LIN {X 0.039,Y -397.005,Z 723.798,A 0.000,B 0.000,C 90.000,E1 179.599} C_DIS
LIN {X 0.011,Y -394.562,Z 723.784,A 0.000,B 0.000,C 90.000,E1 177.135} C_DIS
LIN {X -0.144,Y -391.958,Z 723.766,A 0.000,B 0.000,C 90.000,E1 173.970} C_DIS
LIN {X 0.090,Y -389.994,Z 723.749,A 0.000,B 0.000,C 90.000,E1 170.735} C_DIS
LIN {X -0.181,Y -389.319,Z 723.739,A 0.000,B 0.000,C 90.000,E1 168.993} C_DIS
LIN {X 0.066,Y -388.633,Z 723.729,A 0.000,B 0.000,C 90.000,E1 167.173} C_DIS
LIN {X -0.020,Y -387.919,Z 723.715,A 0.000,B 0.000,C 90.000,E1 164.685} C_DIS
LIN {X -0.021,Y -387.556,Z 723.701,A 0.000,B 0.000,C 90.000,E1 162.181} C_DIS
LIN {X -0.174,Y -387.268,Z 723.687,A 0.000,B 0.000,C 90.000,E1 159.699} C_DIS
LIN {X -0.072,Y -387.127,Z 723.673,A 0.000,B 0.000,C 90.000,E1 157.177} C_DIS
LIN {X -0.029,Y -387.222,Z 723.659,A 0.000,B 0.000,C 90.000,E1 154.665} C_DIS
LIN {X 0.188,Y -387.591,Z 723.643,A 0.000,B 0.000,C 90.000,E1 151.769} C_DIS
LIN {X -0.098,Y -388.115,Z 723.631,A 0.000,B 0.000,C 90.000,E1 149.665} C_DIS
LIN {X 0.077,Y -392.344,Z 723.598,A 0.000,B 0.000,C 90.000,E1 143.577} C_DIS
LIN {X 0.120,Y -395.287,Z 723.584,A 0.000,B 0.000,C 90.000,E1 141.090} C_DIS
LIN {X 0.042,Y -398.011,Z 723.574,A 0.000,B 0.000,C 90.000,E1 139.337} C_DIS
LIN {X -0.158,Y -398.633,Z 723.572,A 0.000,B 0.000,C 90.000,E1 139.013} C_DIS
LIN {X 0.127,Y -401.198,Z 723.566,A 0.000,B 0.000,C 90.000,E1 137.919} C_DIS
LIN {X 0.148,Y -402.865,Z 723.563,A 0.000,B 0.000,C 90.000,E1 137.391} C_DIS
LIN {X -0.092,Y -405.391,Z 723.560,A 0.000,B 0.000,C 90.000,E1 136.863} C_DIS
LIN {X 0.231,Y -408.949,Z 723.557,A 0.000,B 0.000,C 90.000,E1 136.296} C_DIS
LIN {X 0.266,Y -413.856,Z 723.554,A 0.000,B 0.000,C 90.000,E1 135.729} C_DIS
LIN {X 0.176,Y -435.943,Z 723.542,A 0.000,B 0.000,C 90.000,E1 133.542} C_DIS
LIN {X 0.080,Y -449.355,Z 723.535,A 0.000,B 0.000,C 90.000,E1 132.324} C_DIS
LIN {X 0.027,Y -458.279,Z 723.531,A 0.000,B 0.000,C 90.000,E1 131.515} C_DIS
LIN {X -0.130,Y -467.101,Z 723.526,A 0.000,B 0.000,C 90.000,E1 130.701} C_DIS
LIN {X -0.097,Y -474.239,Z 723.522,A 0.000,B 0.000,C 90.000,E1 130.011} C_DIS
LIN {X 0.038,Y -482.703,Z 723.518,A 0.000,B 0.000,C 90.000,E1 129.152} C_DIS
LIN {X -0.057,Y -489.338,Z 723.514,A 0.000,B 0.000,C 90.000,E1 128.463} C_DIS
LIN {X -0.026,Y -496.017,Z 723.510,A 0.000,B 0.000,C 90.000,E1 127.729} C_DIS
LIN {X 0.160,Y -505.000,Z 723.504,A 0.000,B 0.000,C 90.000,E1 126.664} C_DIS
LIN {X 0.076,Y -510.728,Z 723.500,A 0.000,B 0.000,C 90.000,E1 125.931} C_DIS
LIN {X -0.208,Y -513.989,Z 723.497,A 0.000,B 0.000,C 90.000,E1 125.518} C_DIS
LIN {X 0.062,Y -522.250,Z 723.490,A 0.000,B 0.000,C 90.000,E1 124.199} C_DIS
LIN {X -0.204,Y -526.316,Z 723.486,A 0.000,B 0.000,C 90.000,E1 123.499} C_DIS
LIN {X 0.008,Y -530.042,Z 723.482,A 0.000,B 0.000,C 90.000,E1 122.752} C_DIS
LIN {X 0.256,Y -533.521,Z 723.478,A 0.000,B 0.000,C 90.000,E1 122.005} C_DIS
LIN {X -0.198,Y -536.730,Z 723.474,A 0.000,B 0.000,C 90.000,E1 121.337} C_DIS
LIN {X -0.303,Y -541.523,Z 723.468,A 0.000,B 0.000,C 90.000,E1 120.207} C_DIS
LIN {X -0.217,Y -545.563,Z 723.462,A 0.000,B 0.000,C 90.000,E1 119.205} C_DIS
LIN {X 0.272,Y -549.894,Z 723.456,A 0.000,B 0.000,C 90.000,E1 118.025} C_DIS
LIN {X 0.056,Y -552.912,Z 723.451,A 0.000,B 0.000,C 90.000,E1 117.206} C_DIS
LIN {X 0.126,Y -555.717,Z 723.447,A 0.000,B 0.000,C 90.000,E1 116.360} C_DIS
LIN {X -0.023,Y -558.233,Z 723.442,A 0.000,B 0.000,C 90.000,E1 115.540} C_DIS
LIN {X -0.142,Y -560.406,Z 723.437,A 0.000,B 0.000,C 90.000,E1 114.719} C_DIS
LIN {X -0.239,Y -562.322,Z 723.433,A 0.000,B 0.000,C 90.000,E1 113.898} C_DIS
LIN {X 0.200,Y -564.005,Z 723.428,A 0.000,B 0.000,C 90.000,E1 113.025} C_DIS
LIN {X 0.134,Y -565.434,Z 723.423,A 0.000,B 0.000,C 90.000,E1 112.206} C_DIS
LIN {X 0.007,Y -567.636,Z 723.416,A 0.000,B 0.000,C 90.000,E1 110.844} C_DIS
LIN {X 0.250,Y -569.725,Z 723.408,A 0.000,B 0.000,C 90.000,E1 109.450} C_DIS
LIN {X -0.187,Y -571.772,Z 723.401,A 0.000,B 0.000,C 90.000,E1 108.127} C_DIS
LIN {X 0.128,Y -573.658,Z 723.393,A 0.000,B 0.000,C 90.000,E1 106.732} C_DIS
LIN {X -0.210,Y -575.815,Z 723.384,A 0.000,B 0.000,C 90.000,E1 105.134} C_DIS
LIN {X 0.202,Y -577.226,Z 723.378,A 0.000,B 0.000,C 90.000,E1 104.008} C_DIS
LIN {X 0.156,Y -579.651,Z 723.367,A 0.000,B 0.000,C 90.000,E1 102.119} C_DIS
LIN {X 0.032,Y -581.442,Z 723.360,A 0.000,B 0.000,C 90.000,E1 100.782} C_DIS
LIN {X -0.051,Y -583.109,Z 723.352,A 0.000,B 0.000,C 90.000,E1 99.443} C_DIS
LIN {X 0.230,Y -584.312,Z 723.346,A 0.000,B 0.000,C 90.000,E1 98.341} C_DIS
LIN {X -0.234,Y -585.981,Z 723.338,A 0.000,B 0.000,C 90.000,E1 96.777} C_DIS
LIN {X 0.006,Y -587.104,Z 723.332,A 0.000,B 0.000,C 90.000,E1 95.682} C_DIS
LIN {X -0.137,Y -588.453,Z 723.324,A 0.000,B 0.000,C 90.000,E1 94.359} C_DIS
LIN {X -0.264,Y -589.659,Z 723.317,A 0.000,B 0.000,C 90.000,E1 93.037} C_DIS
LIN {X 0.180,Y -590.697,Z 723.309,A 0.000,B 0.000,C 90.000,E1 91.661} C_DIS
LIN {X 0.041,Y -591.560,Z 723.302,A 0.000,B 0.000,C 90.000,E1 90.344} C_DIS
LIN {X -0.082,Y -592.267,Z 723.295,A 0.000,B 0.000,C 90.000,E1 89.026} C_DIS
LIN {X 0.247,Y -592.954,Z 723.284,A 0.000,B 0.000,C 90.000,E1 87.135} C_DIS
LIN {X 0.195,Y -593.220,Z 723.277,A 0.000,B 0.000,C 90.000,E1 85.812} C_DIS
LIN {X 0.157,Y -593.390,Z 723.270,A 0.000,B 0.000,C 90.000,E1 84.489} C_DIS
LIN {X -0.204,Y -593.437,Z 723.261,A 0.000,B 0.000,C 90.000,E1 82.932} C_DIS
LIN {X -0.134,Y -593.361,Z 723.256,A 0.000,B 0.000,C 90.000,E1 82.129} C_DIS
LIN {X -0.028,Y -593.126,Z 723.249,A 0.000,B 0.000,C 90.000,E1 80.792} C_DIS
LIN {X 0.080,Y -592.679,Z 723.242,A 0.000,B 0.000,C 90.000,E1 79.454} C_DIS
LIN {X 0.171,Y -591.925,Z 723.234,A 0.000,B 0.000,C 90.000,E1 78.117} C_DIS
LIN {X -0.117,Y -590.766,Z 723.224,A 0.000,B 0.000,C 90.000,E1 76.284} C_DIS
LIN {X 0.050,Y -589.783,Z 723.216,A 0.000,B 0.000,C 90.000,E1 74.936} C_DIS
LIN {X 0.185,Y -588.443,Z 723.208,A 0.000,B 0.000,C 90.000,E1 73.323} C_DIS
LIN {X -0.361,Y -587.491,Z 723.202,A 0.000,B 0.000,C 90.000,E1 72.308} C_DIS
LIN {X 0.232,Y -586.098,Z 723.194,A 0.000,B 0.000,C 90.000,E1 70.913} C_DIS
LIN {X -0.162,Y -584.968,Z 723.188,A 0.000,B 0.000,C 90.000,E1 69.880} C_DIS
LIN {X -0.167,Y -583.271,Z 723.181,A 0.000,B 0.000,C 90.000,E1 68.539} C_DIS
LIN {X 0.145,Y -581.811,Z 723.175,A 0.000,B 0.000,C 90.000,E1 67.433} C_DIS
LIN {X 0.126,Y -580.195,Z 723.169,A 0.000,B 0.000,C 90.000,E1 66.357} C_DIS
LIN {X 0.096,Y -578.301,Z 723.163,A 0.000,B 0.000,C 90.000,E1 65.281} C_DIS
LIN {X 0.188,Y -576.737,Z 723.158,A 0.000,B 0.000,C 90.000,E1 64.460} C_DIS
LIN {X 0.108,Y -574.431,Z 723.152,A 0.000,B 0.000,C 90.000,E1 63.384} C_DIS
LIN {X 0.149,Y -572.490,Z 723.148,A 0.000,B 0.000,C 90.000,E1 62.564} C_DIS
LIN {X -0.075,Y -570.377,Z 723.143,A 0.000,B 0.000,C 90.000,E1 61.769} C_DIS
LIN {X 0.008,Y -567.228,Z 723.137,A 0.000,B 0.000,C 90.000,E1 60.667} C_DIS
LIN {X -0.261,Y -564.647,Z 723.133,A 0.000,B 0.000,C 90.000,E1 59.871} C_DIS
LIN {X 0.016,Y -560.862,Z 723.126,A 0.000,B 0.000,C 90.000,E1 58.742} C_DIS
LIN {X -0.106,Y -558.780,Z 723.123,A 0.000,B 0.000,C 90.000,E1 58.201} C_DIS
LIN {X -0.242,Y -556.592,Z 723.120,A 0.000,B 0.000,C 90.000,E1 57.661} C_DIS
LIN {X 0.141,Y -552.966,Z 723.116,A 0.000,B 0.000,C 90.000,E1 56.786} C_DIS
LIN {X 0.141,Y -549.488,Z 723.112,A 0.000,B 0.000,C 90.000,E1 56.087} C_DIS
LIN {X 0.218,Y -545.757,Z 723.108,A 0.000,B 0.000,C 90.000,E1 55.388} C_DIS
LIN {X 0.154,Y -541.618,Z 723.104,A 0.000,B 0.000,C 90.000,E1 54.689} C_DIS
LIN {X 0.202,Y -538.072,Z 723.101,A 0.000,B 0.000,C 90.000,E1 54.116} C_DIS
LIN {X -0.090,Y -534.118,Z 723.098,A 0.000,B 0.000,C 90.000,E1 53.577} C_DIS
LIN {X -0.096,Y -529.858,Z 723.094,A 0.000,B 0.000,C 90.000,E1 53.004} C_DIS
LIN {X 0.041,Y -526.322,Z 723.092,A 0.000,B 0.000,C 90.000,E1 52.557} C_DIS
LIN {X 0.213,Y -521.345,Z 723.089,A 0.000,B 0.000,C 90.000,E1 51.984} C_DIS
LIN {X -0.043,Y -515.615,Z 723.086,A 0.000,B 0.000,C 90.000,E1 51.457} C_DIS
LIN {X -0.241,Y -511.106,Z 723.084,A 0.000,B 0.000,C 90.000,E1 51.090} C_DIS
LIN {X 0.069,Y -503.874,Z 723.081,A 0.000,B 0.000,C 90.000,E1 50.481} C_DIS
LIN {X -0.123,Y -498.994,Z 723.079,A 0.000,B 0.000,C 90.000,E1 50.150} C_DIS
LIN {X -0.038,Y -492.505,Z 723.076,A 0.000,B 0.000,C 90.000,E1 49.703} C_DIS
LIN {X 0.015,Y -487.576,Z 723.074,A 0.000,B 0.000,C 90.000,E1 49.380} C_DIS
LIN {X -0.153,Y -471.138,Z 723.069,A 0.000,B 0.000,C 90.000,E1 48.405} C_DIS
LIN {X 0.103,Y -450.074,Z 723.062,A 0.000,B 0.000,C 90.000,E1 47.067} C_DIS
LIN {X -0.031,Y -424.385,Z 723.052,A 0.000,B 0.000,C 90.000,E1 45.364} C_DIS
LIN {X 0.031,Y -419.888,Z 723.050,A 0.000,B 0.000,C 90.000,E1 45.000} C_DIS
LIN {X -0.042,Y -418.828,Z 723.050,A 0.000,B 0.000,C 90.000,E1 44.919} C_DIS
LIN {X -0.072,Y -418.794,Z 723.050,A 0.000,B 0.000,C 90.000,E1 44.919} C_DIS
LIN {X -0.010,Y -415.216,Z 723.041,A 0.000,B 0.000,C 90.000,E1 43.380} C_DIS
LIN {X -0.009,Y -406.545,Z 723.016,A 0.000,B 0.000,C 90.000,E1 38.910} C_DIS
LIN {X 0.137,Y -405.992,Z 723.014,A 0.000,B 0.000,C 90.000,E1 38.543} C_DIS
LIN {X -0.078,Y -406.446,Z 722.995,A 0.000,B 0.000,C 90.000,E1 35.105} C_DIS
LIN {X -0.215,Y -407.693,Z 722.978,A 0.000,B 0.000,C 90.000,E1 32.005} C_DIS
LIN {X 0.110,Y -408.866,Z 722.964,A 0.000,B 0.000,C 90.000,E1 29.539} C_DIS
LIN {X 0.068,Y -410.221,Z 722.951,A 0.000,B 0.000,C 90.000,E1 27.129} C_DIS
LIN {X 0.064,Y -411.807,Z 722.937,A 0.000,B 0.000,C 90.000,E1 24.719} C_DIS
LIN {X 0.183,Y -413.532,Z 722.926,A 0.000,B 0.000,C 90.000,E1 22.642} C_DIS
LIN {X -0.075,Y -416.175,Z 722.911,A 0.000,B 0.000,C 90.000,E1 19.939} C_DIS
LIN {X 0.103,Y -418.796,Z 722.898,A 0.000,B 0.000,C 90.000,E1 17.528} C_DIS
LIN {X 0.181,Y -421.388,Z 722.886,A 0.000,B 0.000,C 90.000,E1 15.481} C_DIS
LIN {X -0.167,Y -423.246,Z 722.879,A 0.000,B 0.000,C 90.000,E1 14.175} C_DIS
LIN {X -0.091,Y -425.603,Z 722.869,A 0.000,B 0.000,C 90.000,E1 12.479} C_DIS
LIN {X -0.176,Y -428.996,Z 722.856,A 0.000,B 0.000,C 90.000,E1 10.141} C_DIS
LIN {X 0.173,Y -432.427,Z 722.843,A 0.000,B 0.000,C 90.000,E1 7.757} C_DIS
LIN {X 0.142,Y -436.373,Z 722.828,A 0.000,B 0.000,C 90.000,E1 5.106} C_DIS
LIN {X -0.160,Y -441.257,Z 722.812,A 0.000,B 0.000,C 90.000,E1 2.178} C_DIS
LIN {X 0.169,Y -445.477,Z 722.799,A 0.000,B 0.000,C 90.000,E1 359.771} C_DIS
LIN {X 0.147,Y -449.319,Z 722.788,A 0.000,B 0.000,C 90.000,E1 357.822} C_DIS
LIN {X -0.138,Y -455.217,Z 722.772,A 0.000,B 0.000,C 90.000,E1 354.951} C_DIS
LIN {X -0.057,Y -458.660,Z 722.763,A 0.000,B 0.000,C 90.000,E1 353.337} C_DIS
LIN {X 0.086,Y -461.964,Z 722.754,A 0.000,B 0.000,C 90.000,E1 351.724} C_DIS
LIN {X -0.032,Y -465.265,Z 722.745,A 0.000,B 0.000,C 90.000,E1 350.151} C_DIS
LIN {X 0.192,Y -468.916,Z 722.735,A 0.000,B 0.000,C 90.000,E1 348.229} C_DIS
LIN {X -0.154,Y -471.771,Z 722.726,A 0.000,B 0.000,C 90.000,E1 346.700} C_DIS
LIN {X -0.042,Y -475.245,Z 722.716,A 0.000,B 0.000,C 90.000,E1 344.810} C_DIS
LIN {X 0.057,Y -481.222,Z 722.698,A 0.000,B 0.000,C 90.000,E1 341.692} C_DIS
LIN {X -0.113,Y -483.295,Z 722.693,A 0.000,B 0.000,C 90.000,E1 340.786} C_DIS
LIN {X 0.191,Y -485.872,Z 722.688,A 0.000,B 0.000,C 90.000,E1 339.826} C_DIS
LIN {X -0.120,Y -488.255,Z 722.685,A 0.000,B 0.000,C 90.000,E1 339.263} C_DIS
LIN {X 0.014,Y -489.779,Z 722.683,A 0.000,B 0.000,C 90.000,E1 338.954} C_DIS
LIN {X 0.287,Y -492.928,Z 722.681,A 0.000,B 0.000,C 90.000,E1 338.465} C_DIS
LIN {X -0.086,Y -495.684,Z 722.679,A 0.000,B 0.000,C 90.000,E1 338.209} C_DIS
LIN {X 0.027,Y -497.240,Z 722.678,A 0.000,B 0.000,C 90.000,E1 338.050} C_DIS
LIN {X 0.041,Y -507.028,Z 722.674,A 0.000,B 0.000,C 90.000,E1 337.283} C_DIS
LIN {X -0.162,Y -527.712,Z 722.666,A 0.000,B 0.000,C 90.000,E1 335.973} C_DIS
LIN {X -0.306,Y -535.606,Z 722.664,A 0.000,B 0.000,C 90.000,E1 335.485} C_DIS
LIN {X 0.031,Y -543.192,Z 722.661,A 0.000,B 0.000,C 90.000,E1 334.921} C_DIS
LIN {X 0.089,Y -548.854,Z 722.658,A 0.000,B 0.000,C 90.000,E1 334.460} C_DIS
LIN {X 0.166,Y -555.938,Z 722.655,A 0.000,B 0.000,C 90.000,E1 333.845} C_DIS
LIN {X -0.262,Y -562.671,Z 722.651,A 0.000,B 0.000,C 90.000,E1 333.256} C_DIS
LIN {X -0.268,Y -569.012,Z 722.648,A 0.000,B 0.000,C 90.000,E1 332.615} C_DIS
LIN {X 0.329,Y -576.355,Z 722.643,A 0.000,B 0.000,C 90.000,E1 331.769} C_DIS
LIN {X 0.023,Y -582.308,Z 722.640,A 0.000,B 0.000,C 90.000,E1 331.129} C_DIS
LIN {X -0.142,Y -590.224,Z 722.634,A 0.000,B 0.000,C 90.000,E1 330.205} C_DIS
LIN {X -0.084,Y -596.782,Z 722.630,A 0.000,B 0.000,C 90.000,E1 329.410} C_DIS
LIN {X 0.197,Y -604.980,Z 722.624,A 0.000,B 0.000,C 90.000,E1 328.329} C_DIS
LIN {X -0.191,Y -610.796,Z 722.620,A 0.000,B 0.000,C 90.000,E1 327.582} C_DIS
LIN {X 0.011,Y -615.420,Z 722.616,A 0.000,B 0.000,C 90.000,E1 326.914} C_DIS
LIN {X -0.264,Y -619.801,Z 722.613,A 0.000,B 0.000,C 90.000,E1 326.294} C_DIS
LIN {X -0.165,Y -624.737,Z 722.608,A 0.000,B 0.000,C 90.000,E1 325.515} C_DIS
LIN {X -0.009,Y -629.428,Z 722.604,A 0.000,B 0.000,C 90.000,E1 324.736} C_DIS
LIN {X 0.200,Y -634.627,Z 722.599,A 0.000,B 0.000,C 90.000,E1 323.829} C_DIS
LIN {X -0.041,Y -640.211,Z 722.594,A 0.000,B 0.000,C 90.000,E1 322.844} C_DIS
LIN {X 0.186,Y -646.095,Z 722.587,A 0.000,B 0.000,C 90.000,E1 321.698} C_DIS
LIN {X -0.039,Y -650.451,Z 722.583,A 0.000,B 0.000,C 90.000,E1 320.848} C_DIS
LIN {X -0.133,Y -653.989,Z 722.578,A 0.000,B 0.000,C 90.000,E1 320.114} C_DIS
LIN {X 0.253,Y -658.472,Z 722.573,A 0.000,B 0.000,C 90.000,E1 319.094} C_DIS
LIN {X -0.302,Y -662.697,Z 722.567,A 0.000,B 0.000,C 90.000,E1 318.162} C_DIS
LIN {X 0.133,Y -667.465,Z 722.561,A 0.000,B 0.000,C 90.000,E1 316.905} C_DIS
LIN {X -0.311,Y -670.969,Z 722.555,A 0.000,B 0.000,C 90.000,E1 315.972} C_DIS
LIN {X -0.245,Y -674.306,Z 722.550,A 0.000,B 0.000,C 90.000,E1 315.000} C_DIS
LIN {X -0.137,Y -677.375,Z 722.545,A 0.000,B 0.000,C 90.000,E1 314.028} C_DIS
LIN {X 0.046,Y -681.033,Z 722.538,A 0.000,B 0.000,C 90.000,E1 312.813} C_DIS
LIN {X 0.273,Y -683.745,Z 722.533,A 0.000,B 0.000,C 90.000,E1 311.838} C_DIS
LIN {X -0.025,Y -685.667,Z 722.529,A 0.000,B 0.000,C 90.000,E1 311.148} C_DIS
LIN {X 0.332,Y -688.548,Z 722.522,A 0.000,B 0.000,C 90.000,E1 309.930} C_DIS
LIN {X -0.369,Y -690.082,Z 722.518,A 0.000,B 0.000,C 90.000,E1 309.277} C_DIS
LIN {X -0.019,Y -691.864,Z 722.513,A 0.000,B 0.000,C 90.000,E1 308.302} C_DIS
LIN {X -0.078,Y -693.389,Z 722.508,A 0.000,B 0.000,C 90.000,E1 307.363} C_DIS
LIN {X -0.121,Y -694.713,Z 722.502,A 0.000,B 0.000,C 90.000,E1 306.423} C_DIS
LIN {X 0.008,Y -695.901,Z 722.497,A 0.000,B 0.000,C 90.000,E1 305.471} C_DIS
LIN {X -0.008,Y -696.862,Z 722.492,A 0.000,B 0.000,C 90.000,E1 304.532} C_DIS
LIN {X 0.104,Y -698.338,Z 722.483,A 0.000,B 0.000,C 90.000,E1 302.880} C_DIS
LIN {X 0.209,Y -699.491,Z 722.475,A 0.000,B 0.000,C 90.000,E1 301.465} C_DIS
LIN {X -0.210,Y -700.017,Z 722.471,A 0.000,B 0.000,C 90.000,E1 300.797} C_DIS
LIN {X -0.018,Y -700.369,Z 722.467,A 0.000,B 0.000,C 90.000,E1 300.079} C_DIS
LIN {X 0.113,Y -700.721,Z 722.461,A 0.000,B 0.000,C 90.000,E1 298.899} C_DIS
LIN {X 0.177,Y -701.185,Z 722.452,A 0.000,B 0.000,C 90.000,E1 297.257} C_DIS
LIN {X -0.091,Y -701.933,Z 722.442,A 0.000,B 0.000,C 90.000,E1 295.643} C_DIS
LIN {X 0.162,Y -702.111,Z 722.440,A 0.000,B 0.000,C 90.000,E1 295.155} C_DIS
LIN {X -0.215,Y -701.889,Z 722.437,A 0.000,B 0.000,C 90.000,E1 294.719} C_DIS
LIN {X 0.063,Y -701.608,Z 722.436,A 0.000,B 0.000,C 90.000,E1 294.463} C_DIS
LIN {X 0.339,Y -700.851,Z 722.435,A 0.000,B 0.000,C 90.000,E1 294.207} C_DIS
LIN {X -0.028,Y -699.929,Z 722.433,A 0.000,B 0.000,C 90.000,E1 294.003} C_DIS
LIN {X -0.040,Y -698.772,Z 722.432,A 0.000,B 0.000,C 90.000,E1 293.770} C_DIS
LIN {X 0.092,Y -697.749,Z 722.431,A 0.000,B 0.000,C 90.000,E1 293.643} C_DIS
LIN {X -0.208,Y -693.584,Z 722.430,A 0.000,B 0.000,C 90.000,E1 293.334} C_DIS
LIN {X 0.100,Y -692.207,Z 722.429,A 0.000,B 0.000,C 90.000,E1 293.206} C_DIS
LIN {X -0.228,Y -690.549,Z 722.428,A 0.000,B 0.000,C 90.000,E1 293.131} C_DIS
LIN {X -0.252,Y -685.626,Z 722.427,A 0.000,B 0.000,C 90.000,E1 292.950} C_DIS
LIN {X 0.155,Y -677.566,Z 722.426,A 0.000,B 0.000,C 90.000,E1 292.717} C_DIS
LIN {X -0.157,Y -665.539,Z 722.425,A 0.000,B 0.000,C 90.000,E1 292.589} C_DIS
LIN {X 0.226,Y -653.406,Z 722.424,A 0.000,B 0.000,C 90.000,E1 292.386} C_DIS
LIN {X 0.360,Y -643.395,Z 722.424,A 0.000,B 0.000,C 90.000,E1 292.206} C_DIS
LIN {X 0.111,Y -633.310,Z 722.422,A 0.000,B 0.000,C 90.000,E1 292.025} C_DIS
LIN {X -0.014,Y -619.796,Z 722.421,A 0.000,B 0.000,C 90.000,E1 291.716} C_DIS
LIN {X 0.084,Y -585.271,Z 722.415,A 0.000,B 0.000,C 90.000,E1 290.737} C_DIS
LIN {X 0.041,Y -572.684,Z 722.413,A 0.000,B 0.000,C 90.000,E1 290.375} C_DIS
LIN {X -0.158,Y -567.427,Z 722.412,A 0.000,B 0.000,C 90.000,E1 290.248} C_DIS
LIN {X -0.326,Y -561.712,Z 722.411,A 0.000,B 0.000,C 90.000,E1 290.066} C_DIS
LIN {X -0.192,Y -560.293,Z 722.411,A 0.000,B 0.000,C 90.000,E1 289.993} C_DIS
LIN {X 0.174,Y -556.366,Z 722.410,A 0.000,B 0.000,C 90.000,E1 289.704} C_DIS
LIN {X 0.144,Y -556.323,Z 722.410,A 0.000,B 0.000,C 90.000,E1 289.704} C_DIS
LIN {X -0.230,Y -555.487,Z 722.409,A 0.000,B 0.000,C 90.000,E1 289.577} C_DIS
LIN {X -0.210,Y -554.790,Z 722.406,A 0.000,B 0.000,C 90.000,E1 289.087} C_DIS
LIN {X 0.223,Y -554.436,Z 722.400,A 0.000,B 0.000,C 90.000,E1 288.000} C_DIS
LIN {X -0.092,Y -553.662,Z 722.389,A 0.000,B 0.000,C 90.000,E1 286.079} C_DIS
LIN {X -0.052,Y -552.976,Z 722.378,A 0.000,B 0.000,C 90.000,E1 284.120} C_DIS
LIN {X -0.171,Y -552.369,Z 722.368,A 0.000,B 0.000,C 90.000,E1 282.175} C_DIS
LIN {X 0.009,Y -551.561,Z 722.357,A 0.000,B 0.000,C 90.000,E1 280.197} C_DIS
LIN {X -0.050,Y -550.911,Z 722.349,A 0.000,B 0.000,C 90.000,E1 278.803} C_DIS
LIN {X 0.010,Y -549.980,Z 722.338,A 0.000,B 0.000,C 90.000,E1 276.834} C_DIS
LIN {X -0.078,Y -549.286,Z 722.327,A 0.000,B 0.000,C 90.000,E1 274.878} C_DIS
LIN {X 0.188,Y -548.942,Z 722.321,A 0.000,B 0.000,C 90.000,E1 273.726} C_DIS
LIN {X -0.089,Y -548.386,Z 722.313,A 0.000,B 0.000,C 90.000,E1 272.350} C_DIS
LIN {X 0.121,Y -547.957,Z 722.307,A 0.000,B 0.000,C 90.000,E1 271.203} C_DIS
LIN {X -0.235,Y -547.342,Z 722.301,A 0.000,B 0.000,C 90.000,E1 270.115} C_DIS
LIN {X 0.035,Y -546.339,Z 722.291,A 0.000,B 0.000,C 90.000,E1 268.396} C_DIS
LIN {X -0.230,Y -545.264,Z 722.282,A 0.000,B 0.000,C 90.000,E1 266.731} C_DIS
LIN {X -0.034,Y -544.270,Z 722.274,A 0.000,B 0.000,C 90.000,E1 265.298} C_DIS
LIN {X 0.245,Y -543.040,Z 722.264,A 0.000,B 0.000,C 90.000,E1 263.571} C_DIS
LIN {X -0.050,Y -541.883,Z 722.257,A 0.000,B 0.000,C 90.000,E1 262.186} C_DIS
LIN {X -0.212,Y -540.424,Z 722.247,A 0.000,B 0.000,C 90.000,E1 260.500} C_DIS
LIN {X 0.129,Y -538.917,Z 722.238,A 0.000,B 0.000,C 90.000,E1 258.757} C_DIS
LIN {X -0.061,Y -537.725,Z 722.230,A 0.000,B 0.000,C 90.000,E1 257.353} C_DIS
LIN {X -0.152,Y -536.482,Z 722.222,A 0.000,B 0.000,C 90.000,E1 255.936} C_DIS
LIN {X -0.266,Y -535.008,Z 722.214,A 0.000,B 0.000,C 90.000,E1 254.519} C_DIS
LIN {X -0.074,Y -533.236,Z 722.204,A 0.000,B 0.000,C 90.000,E1 252.779} C_DIS
LIN {X 0.057,Y -531.784,Z 722.196,A 0.000,B 0.000,C 90.000,E1 251.329} C_DIS
LIN {X -0.041,Y -530.735,Z 722.192,A 0.000,B 0.000,C 90.000,E1 250.477} C_DIS
LIN {X 0.219,Y -528.473,Z 722.182,A 0.000,B 0.000,C 90.000,E1 248.720} C_DIS
LIN {X -0.038,Y -526.823,Z 722.176,A 0.000,B 0.000,C 90.000,E1 247.592} C_DIS
LIN {X 0.131,Y -524.659,Z 722.167,A 0.000,B 0.000,C 90.000,E1 246.125} C_DIS
LIN {X 0.195,Y -522.292,Z 722.159,A 0.000,B 0.000,C 90.000,E1 244.665} C_DIS
LIN {X 0.078,Y -520.376,Z 722.153,A 0.000,B 0.000,C 90.000,E1 243.512} C_DIS
LIN {X -0.067,Y -518.223,Z 722.146,A 0.000,B 0.000,C 90.000,E1 242.359} C_DIS
LIN {X 0.020,Y -514.745,Z 722.137,A 0.000,B 0.000,C 90.000,E1 240.589} C_DIS
LIN {X 0.032,Y -512.370,Z 722.130,A 0.000,B 0.000,C 90.000,E1 239.410} C_DIS
LIN {X -0.197,Y -508.678,Z 722.120,A 0.000,B 0.000,C 90.000,E1 237.661} C_DIS
LIN {X -0.232,Y -504.945,Z 722.110,A 0.000,B 0.000,C 90.000,E1 235.881} C_DIS
LIN {X -0.251,Y -502.230,Z 722.104,A 0.000,B 0.000,C 90.000,E1 234.689} C_DIS
LIN {X -0.191,Y -500.109,Z 722.099,A 0.000,B 0.000,C 90.000,E1 233.783} C_DIS
LIN {X 0.264,Y -498.652,Z 722.095,A 0.000,B 0.000,C 90.000,E1 233.130} C_DIS
LIN {X 0.186,Y -492.482,Z 722.082,A 0.000,B 0.000,C 90.000,E1 230.723} C_DIS
LIN {X -0.139,Y -486.788,Z 722.068,A 0.000,B 0.000,C 90.000,E1 228.324} C_DIS
LIN {X 0.120,Y -483.977,Z 722.062,A 0.000,B 0.000,C 90.000,E1 227.067} C_DIS
LIN {X -0.086,Y -479.841,Z 722.051,A 0.000,B 0.000,C 90.000,E1 225.243} C_DIS
LIN {X 0.054,Y -475.180,Z 722.039,A 0.000,B 0.000,C 90.000,E1 223.056} C_DIS
LIN {X -0.010,Y -471.250,Z 722.029,A 0.000,B 0.000,C 90.000,E1 221.191} C_DIS
LIN {X -0.185,Y -467.848,Z 722.020,A 0.000,B 0.000,C 90.000,E1 219.644} C_DIS
LIN {X 0.237,Y -464.333,Z 722.011,A 0.000,B 0.000,C 90.000,E1 218.016} C_DIS
LIN {X 0.012,Y -458.170,Z 721.996,A 0.000,B 0.000,C 90.000,E1 215.185} C_DIS
LIN {X -0.113,Y -453.927,Z 721.983,A 0.000,B 0.000,C 90.000,E1 212.959} C_DIS
LIN {X -0.148,Y -449.164,Z 721.969,A 0.000,B 0.000,C 90.000,E1 210.384} C_DIS
LIN {X 0.006,Y -446.100,Z 721.960,A 0.000,B 0.000,C 90.000,E1 208.743} C_DIS
LIN {X -0.059,Y -442.596,Z 721.949,A 0.000,B 0.000,C 90.000,E1 206.796} C_DIS
LIN {X 0.114,Y -440.139,Z 721.942,A 0.000,B 0.000,C 90.000,E1 205.463} C_DIS
LIN {X 0.082,Y -437.170,Z 721.932,A 0.000,B 0.000,C 90.000,E1 203.823} C_DIS
LIN {X 0.048,Y -433.493,Z 721.921,A 0.000,B 0.000,C 90.000,E1 201.844} C_DIS
LIN {X 0.112,Y -430.395,Z 721.912,A 0.000,B 0.000,C 90.000,E1 200.174} C_DIS
LIN {X 0.022,Y -426.783,Z 721.901,A 0.000,B 0.000,C 90.000,E1 198.181} C_DIS
LIN {X 0.133,Y -422.996,Z 721.890,A 0.000,B 0.000,C 90.000,E1 196.150} C_DIS
LIN {X -0.200,Y -418.730,Z 721.877,A 0.000,B 0.000,C 90.000,E1 193.828} C_DIS
LIN {X -0.041,Y -414.501,Z 721.863,A 0.000,B 0.000,C 90.000,E1 191.422} C_DIS
LIN {X -0.091,Y -410.285,Z 721.850,A 0.000,B 0.000,C 90.000,E1 189.029} C_DIS
LIN {X -0.041,Y -406.502,Z 721.837,A 0.000,B 0.000,C 90.000,E1 186.606} C_DIS
LIN {X -0.130,Y -402.880,Z 721.823,A 0.000,B 0.000,C 90.000,E1 184.188} C_DIS
LIN {X 0.116,Y -400.484,Z 721.814,A 0.000,B 0.000,C 90.000,E1 182.407} C_DIS
LIN {X 0.187,Y -397.519,Z 721.800,A 0.000,B 0.000,C 90.000,E1 179.943} C_DIS
LIN {X 0.106,Y -394.684,Z 721.784,A 0.000,B 0.000,C 90.000,E1 177.135} C_DIS
LIN {X -0.045,Y -392.108,Z 721.767,A 0.000,B 0.000,C 90.000,E1 173.970} C_DIS
LIN {X -0.190,Y -390.172,Z 721.749,A 0.000,B 0.000,C 90.000,E1 170.792} C_DIS
LIN {X -0.073,Y -389.474,Z 721.739,A 0.000,B 0.000,C 90.000,E1 168.993} C_DIS
LIN {X -0.227,Y -388.968,Z 721.731,A 0.000,B 0.000,C 90.000,E1 167.589} C_DIS
LIN {X 0.066,Y -388.261,Z 721.717,A 0.000,B 0.000,C 90.000,E1 165.046} C_DIS
LIN {X 0.102,Y -387.775,Z 721.701,A 0.000,B 0.000,C 90.000,E1 162.181} C_DIS
LIN {X -0.075,Y -387.523,Z 721.689,A 0.000,B 0.000,C 90.000,E1 160.061} C_DIS
LIN {X 0.041,Y -387.386,Z 721.675,A 0.000,B 0.000,C 90.000,E1 157.539} C_DIS
LIN {X -0.062,Y -387.463,Z 721.661,A 0.000,B 0.000,C 90.000,E1 155.049} C_DIS
LIN {X -0.020,Y -387.736,Z 721.647,A 0.000,B 0.000,C 90.000,E1 152.538} C_DIS
LIN {X 0.040,Y -388.186,Z 721.636,A 0.000,B 0.000,C 90.000,E1 150.383} C_DIS
LIN {X 0.053,Y -390.003,Z 721.614,A 0.000,B 0.000,C 90.000,E1 146.453} C_DIS
LIN {X 0.207,Y -394.899,Z 721.586,A 0.000,B 0.000,C 90.000,E1 141.457} C_DIS
LIN {X 0.122,Y -397.333,Z 721.576,A 0.000,B 0.000,C 90.000,E1 139.703} C_DIS
LIN {X 0.021,Y -398.511,Z 721.572,A 0.000,B 0.000,C 90.000,E1 139.013} C_DIS
LIN {X 0.037,Y -400.807,Z 721.567,A 0.000,B 0.000,C 90.000,E1 137.957} C_DIS
LIN {X -0.127,Y -402.523,Z 721.563,A 0.000,B 0.000,C 90.000,E1 137.391} C_DIS
LIN {X -0.100,Y -404.795,Z 721.560,A 0.000,B 0.000,C 90.000,E1 136.863} C_DIS
LIN {X 0.090,Y -405.666,Z 721.559,A 0.000,B 0.000,C 90.000,E1 136.662} C_DIS
LIN {X 0.145,Y -409.207,Z 721.556,A 0.000,B 0.000,C 90.000,E1 136.134} C_DIS
LIN {X -0.163,Y -413.747,Z 721.554,A 0.000,B 0.000,C 90.000,E1 135.648} C_DIS
LIN {X -0.044,Y -426.310,Z 721.546,A 0.000,B 0.000,C 90.000,E1 134.352} C_DIS
LIN {X 0.038,Y -448.773,Z 721.535,A 0.000,B 0.000,C 90.000,E1 132.243} C_DIS
LIN {X -0.095,Y -459.211,Z 721.529,A 0.000,B 0.000,C 90.000,E1 131.310} C_DIS
LIN {X 0.158,Y -467.951,Z 721.525,A 0.000,B 0.000,C 90.000,E1 130.458} C_DIS
LIN {X 0.037,Y -473.658,Z 721.522,A 0.000,B 0.000,C 90.000,E1 129.930} C_DIS
LIN {X -0.174,Y -482.132,Z 721.517,A 0.000,B 0.000,C 90.000,E1 129.116} C_DIS
LIN {X -0.124,Y -487.561,Z 721.514,A 0.000,B 0.000,C 90.000,E1 128.543} C_DIS
LIN {X 0.092,Y -495.651,Z 721.509,A 0.000,B 0.000,C 90.000,E1 127.649} C_DIS
LIN {X 0.057,Y -504.273,Z 721.504,A 0.000,B 0.000,C 90.000,E1 126.664} C_DIS
LIN {X 0.129,Y -510.005,Z 721.500,A 0.000,B 0.000,C 90.000,E1 125.931} C_DIS
LIN {X -0.221,Y -514.195,Z 721.497,A 0.000,B 0.000,C 90.000,E1 125.391} C_DIS
LIN {X 0.209,Y -519.082,Z 721.492,A 0.000,B 0.000,C 90.000,E1 124.612} C_DIS
LIN {X -0.026,Y -521.906,Z 721.490,A 0.000,B 0.000,C 90.000,E1 124.199} C_DIS
LIN {X 0.143,Y -526.053,Z 721.486,A 0.000,B 0.000,C 90.000,E1 123.452} C_DIS
LIN {X -0.086,Y -529.849,Z 721.482,A 0.000,B 0.000,C 90.000,E1 122.752} C_DIS
LIN {X 0.061,Y -532.760,Z 721.479,A 0.000,B 0.000,C 90.000,E1 122.163} C_DIS
LIN {X -0.263,Y -536.625,Z 721.474,A 0.000,B 0.000,C 90.000,E1 121.337} C_DIS
LIN {X 0.237,Y -542.090,Z 721.467,A 0.000,B 0.000,C 90.000,E1 120.001} C_DIS
LIN {X -0.048,Y -547.749,Z 721.459,A 0.000,B 0.000,C 90.000,E1 118.615} C_DIS
LIN {X -0.034,Y -550.945,Z 721.454,A 0.000,B 0.000,C 90.000,E1 117.769} C_DIS
LIN {X 0.280,Y -554.860,Z 721.448,A 0.000,B 0.000,C 90.000,E1 116.616} C_DIS
LIN {X 0.123,Y -557.479,Z 721.443,A 0.000,B 0.000,C 90.000,E1 115.796} C_DIS
LIN {X -0.003,Y -559.806,Z 721.439,A 0.000,B 0.000,C 90.000,E1 114.975} C_DIS
LIN {X 0.126,Y -561.856,Z 721.434,A 0.000,B 0.000,C 90.000,E1 114.131} C_DIS
LIN {X -0.187,Y -563.649,Z 721.430,A 0.000,B 0.000,C 90.000,E1 113.334} C_DIS
LIN {X 0.266,Y -565.193,Z 721.425,A 0.000,B 0.000,C 90.000,E1 112.461} C_DIS
LIN {X -0.052,Y -567.866,Z 721.416,A 0.000,B 0.000,C 90.000,E1 110.844} C_DIS
LIN {X -0.186,Y -570.395,Z 721.407,A 0.000,B 0.000,C 90.000,E1 109.214} C_DIS
LIN {X -0.238,Y -572.062,Z 721.401,A 0.000,B 0.000,C 90.000,E1 108.127} C_DIS
LIN {X 0.082,Y -573.957,Z 721.393,A 0.000,B 0.000,C 90.000,E1 106.732} C_DIS
LIN {X 0.102,Y -576.517,Z 721.383,A 0.000,B 0.000,C 90.000,E1 104.828} C_DIS
LIN {X 0.167,Y -577.591,Z 721.378,A 0.000,B 0.000,C 90.000,E1 104.008} C_DIS
LIN {X 0.131,Y -580.046,Z 721.367,A 0.000,B 0.000,C 90.000,E1 102.119} C_DIS
LIN {X 0.014,Y -581.867,Z 721.360,A 0.000,B 0.000,C 90.000,E1 100.782} C_DIS
LIN {X -0.063,Y -583.547,Z 721.352,A 0.000,B 0.000,C 90.000,E1 99.443} C_DIS
LIN {X 0.225,Y -584.781,Z 721.346,A 0.000,B 0.000,C 90.000,E1 98.341} C_DIS
LIN {X 0.008,Y -586.763,Z 721.336,A 0.000,B 0.000,C 90.000,E1 96.486} C_DIS
LIN {X -0.146,Y -588.123,Z 721.329,A 0.000,B 0.000,C 90.000,E1 95.163} C_DIS
LIN {X -0.275,Y -589.453,Z 721.321,A 0.000,B 0.000,C 90.000,E1 93.841} C_DIS
LIN {X 0.169,Y -590.610,Z 721.314,A 0.000,B 0.000,C 90.000,E1 92.465} C_DIS
LIN {X 0.044,Y -591.601,Z 721.306,A 0.000,B 0.000,C 90.000,E1 91.146} C_DIS
LIN {X -0.078,Y -592.405,Z 721.299,A 0.000,B 0.000,C 90.000,E1 89.828} C_DIS
LIN {X 0.189,Y -592.923,Z 721.293,A 0.000,B 0.000,C 90.000,E1 88.740} C_DIS
LIN {X -0.277,Y -593.498,Z 721.284,A 0.000,B 0.000,C 90.000,E1 87.192} C_DIS
LIN {X 0.274,Y -593.765,Z 721.277,A 0.000,B 0.000,C 90.000,E1 85.812} C_DIS
LIN {X -0.139,Y -593.956,Z 721.268,A 0.000,B 0.000,C 90.000,E1 84.261} C_DIS
LIN {X 0.092,Y -593.941,Z 721.259,A 0.000,B 0.000,C 90.000,E1 82.648} C_DIS
LIN {X 0.120,Y -593.745,Z 721.252,A 0.000,B 0.000,C 90.000,E1 81.319} C_DIS
LIN {X -0.045,Y -593.448,Z 721.246,A 0.000,B 0.000,C 90.000,E1 80.274} C_DIS
LIN {X -0.103,Y -593.012,Z 721.240,A 0.000,B 0.000,C 90.000,E1 79.218} C_DIS
LIN {X -0.006,Y -592.204,Z 721.233,A 0.000,B 0.000,C 90.000,E1 77.881} C_DIS
LIN {X 0.291,Y -590.987,Z 721.222,A 0.000,B 0.000,C 90.000,E1 75.992} C_DIS
LIN {X 0.300,Y -589.723,Z 721.214,A 0.000,B 0.000,C 90.000,E1 74.393} C_DIS
LIN {X -0.123,Y -588.324,Z 721.205,A 0.000,B 0.000,C 90.000,E1 72.834} C_DIS
LIN {X -0.109,Y -587.267,Z 721.199,A 0.000,B 0.000,C 90.000,E1 71.764} C_DIS
LIN {X 0.143,Y -585.525,Z 721.190,A 0.000,B 0.000,C 90.000,E1 70.134} C_DIS
LIN {X -0.057,Y -584.252,Z 721.184,A 0.000,B 0.000,C 90.000,E1 69.082} C_DIS
LIN {X 0.141,Y -582.431,Z 721.176,A 0.000,B 0.000,C 90.000,E1 67.720} C_DIS
LIN {X 0.304,Y -580.381,Z 721.169,A 0.000,B 0.000,C 90.000,E1 66.357} C_DIS
LIN {X 0.033,Y -578.436,Z 721.163,A 0.000,B 0.000,C 90.000,E1 65.305} C_DIS
LIN {X 0.120,Y -576.825,Z 721.158,A 0.000,B 0.000,C 90.000,E1 64.485} C_DIS
LIN {X 0.290,Y -574.472,Z 721.152,A 0.000,B 0.000,C 90.000,E1 63.384} C_DIS
LIN {X -0.178,Y -572.462,Z 721.148,A 0.000,B 0.000,C 90.000,E1 62.615} C_DIS
LIN {X 0.105,Y -570.350,Z 721.143,A 0.000,B 0.000,C 90.000,E1 61.769} C_DIS
LIN {X 0.186,Y -567.166,Z 721.137,A 0.000,B 0.000,C 90.000,E1 60.667} C_DIS
LIN {X 0.010,Y -563.558,Z 721.131,A 0.000,B 0.000,C 90.000,E1 59.587} C_DIS
LIN {X 0.189,Y -560.683,Z 721.127,A 0.000,B 0.000,C 90.000,E1 58.742} C_DIS
LIN {X 0.147,Y -557.428,Z 721.122,A 0.000,B 0.000,C 90.000,E1 57.916} C_DIS
LIN {X 0.003,Y -555.053,Z 721.119,A 0.000,B 0.000,C 90.000,E1 57.375} C_DIS
LIN {X -0.158,Y -552.588,Z 721.116,A 0.000,B 0.000,C 90.000,E1 56.834} C_DIS
LIN {X -0.159,Y -549.023,Z 721.112,A 0.000,B 0.000,C 90.000,E1 56.135} C_DIS
LIN {X 0.261,Y -545.105,Z 721.108,A 0.000,B 0.000,C 90.000,E1 55.388} C_DIS
LIN {X 0.021,Y -541.782,Z 721.105,A 0.000,B 0.000,C 90.000,E1 54.848} C_DIS
LIN {X 0.102,Y -538.266,Z 721.102,A 0.000,B 0.000,C 90.000,E1 54.276} C_DIS
LIN {X 0.125,Y -534.305,Z 721.098,A 0.000,B 0.000,C 90.000,E1 53.703} C_DIS
LIN {X -0.268,Y -530.294,Z 721.096,A 0.000,B 0.000,C 90.000,E1 53.210} C_DIS
LIN {X 0.014,Y -525.792,Z 721.092,A 0.000,B 0.000,C 90.000,E1 52.637} C_DIS
LIN {X -0.069,Y -520.904,Z 721.089,A 0.000,B 0.000,C 90.000,E1 52.110} C_DIS
LIN {X 0.228,Y -515.272,Z 721.086,A 0.000,B 0.000,C 90.000,E1 51.537} C_DIS
LIN {X 0.043,Y -509.093,Z 721.084,A 0.000,B 0.000,C 90.000,E1 51.045} C_DIS
LIN {X 0.106,Y -502.889,Z 721.081,A 0.000,B 0.000,C 90.000,E1 50.561} C_DIS
LIN {X 0.027,Y -498.139,Z 721.079,A 0.000,B 0.000,C 90.000,E1 50.231} C_DIS
LIN {X -0.090,Y -489.988,Z 721.076,A 0.000,B 0.000,C 90.000,E1 49.703} C_DIS
LIN {X 0.116,Y -481.722,Z 721.073,A 0.000,B 0.000,C 90.000,E1 49.175} C_DIS
LIN {X 0.152,Y -463.698,Z 721.067,A 0.000,B 0.000,C 90.000,E1 48.081} C_DIS
LIN {X 0.004,Y -434.307,Z 721.057,A 0.000,B 0.000,C 90.000,E1 46.215} C_DIS
LIN {X -0.076,Y -424.735,Z 721.053,A 0.000,B 0.000,C 90.000,E1 45.567} C_DIS
LIN {X 0.046,Y -419.797,Z 721.051,A 0.000,B 0.000,C 90.000,E1 45.162} C_DIS
LIN {X 0.225,Y -419.162,Z 721.051,A 0.000,B 0.000,C 90.000,E1 45.081} C_DIS
LIN {X 0.196,Y -419.138,Z 721.051,A 0.000,B 0.000,C 90.000,E1 45.081} C_DIS
LIN {X 0.154,Y -418.710,Z 721.049,A 0.000,B 0.000,C 90.000,E1 44.838} C_DIS
LIN {X -0.221,Y -409.314,Z 721.025,A 0.000,B 0.000,C 90.000,E1 40.539} C_DIS
LIN {X 0.224,Y -406.339,Z 721.016,A 0.000,B 0.000,C 90.000,E1 38.749} C_DIS
LIN {X 0.019,Y -406.788,Z 720.996,A 0.000,B 0.000,C 90.000,E1 35.311} C_DIS
LIN {X -0.106,Y -408.019,Z 720.979,A 0.000,B 0.000,C 90.000,E1 32.212} C_DIS
LIN {X -0.122,Y -409.197,Z 720.965,A 0.000,B 0.000,C 90.000,E1 29.795} C_DIS
LIN {X -0.159,Y -410.534,Z 720.952,A 0.000,B 0.000,C 90.000,E1 27.385} C_DIS
LIN {X 0.137,Y -412.346,Z 720.937,A 0.000,B 0.000,C 90.000,E1 24.591} C_DIS
LIN {X -0.115,Y -414.074,Z 720.925,A 0.000,B 0.000,C 90.000,E1 22.567} C_DIS
LIN {X 0.024,Y -416.726,Z 720.910,A 0.000,B 0.000,C 90.000,E1 19.812} C_DIS
LIN {X -0.186,Y -419.365,Z 720.897,A 0.000,B 0.000,C 90.000,E1 17.457} C_DIS
LIN {X -0.047,Y -422.434,Z 720.884,A 0.000,B 0.000,C 90.000,E1 15.064} C_DIS
LIN {X -0.048,Y -425.665,Z 720.871,A 0.000,B 0.000,C 90.000,E1 12.703} C_DIS
LIN {X -0.145,Y -429.034,Z 720.858,A 0.000,B 0.000,C 90.000,E1 10.366} C_DIS
LIN {X -0.177,Y -432.888,Z 720.843,A 0.000,B 0.000,C 90.000,E1 7.701} C_DIS
LIN {X -0.194,Y -436.828,Z 720.828,A 0.000,B 0.000,C 90.000,E1 5.049} C_DIS
LIN {X -0.040,Y -441.707,Z 720.811,A 0.000,B 0.000,C 90.000,E1 2.064} C_DIS
LIN {X 0.169,Y -445.722,Z 720.799,A 0.000,B 0.000,C 90.000,E1 359.771} C_DIS
LIN {X 0.153,Y -449.561,Z 720.788,A 0.000,B 0.000,C 90.000,E1 357.822} C_DIS
LIN {X -0.124,Y -455.413,Z 720.772,A 0.000,B 0.000,C 90.000,E1 354.951} C_DIS
LIN {X -0.039,Y -458.857,Z 720.763,A 0.000,B 0.000,C 90.000,E1 353.337} C_DIS
LIN {X 0.108,Y -462.129,Z 720.754,A 0.000,B 0.000,C 90.000,E1 351.724} C_DIS
LIN {X 0.193,Y -464.796,Z 720.747,A 0.000,B 0.000,C 90.000,E1 350.443} C_DIS
LIN {X 0.061,Y -466.631,Z 720.742,A 0.000,B 0.000,C 90.000,E1 349.511} C_DIS
LIN {X 0.036,Y -469.650,Z 720.733,A 0.000,B 0.000,C 90.000,E1 347.937} C_DIS
LIN {X -0.015,Y -473.057,Z 720.723,A 0.000,B 0.000,C 90.000,E1 346.061} C_DIS
LIN {X -0.176,Y -475.947,Z 720.714,A 0.000,B 0.000,C 90.000,E1 344.519} C_DIS
LIN {X 0.099,Y -481.348,Z 720.698,A 0.000,B 0.000,C 90.000,E1 341.692} C_DIS
LIN {X -0.069,Y -484.053,Z 720.692,A 0.000,B 0.000,C 90.000,E1 340.477} C_DIS
LIN {X -0.222,Y -485.700,Z 720.688,A 0.000,B 0.000,C 90.000,E1 339.880} C_DIS
LIN {X -0.212,Y -486.618,Z 720.686,A 0.000,B 0.000,C 90.000,E1 339.571} C_DIS
LIN {X 0.096,Y -488.331,Z 720.684,A 0.000,B 0.000,C 90.000,E1 339.082} C_DIS
LIN {X -0.008,Y -491.004,Z 720.681,A 0.000,B 0.000,C 90.000,E1 338.592} C_DIS
LIN {X 0.024,Y -493.123,Z 720.679,A 0.000,B 0.000,C 90.000,E1 338.284} C_DIS
LIN {X -0.020,Y -497.335,Z 720.677,A 0.000,B 0.000,C 90.000,E1 337.847} C_DIS
LIN {X 0.005,Y -502.597,Z 720.675,A 0.000,B 0.000,C 90.000,E1 337.411} C_DIS
LIN {X -0.034,Y -508.587,Z 720.672,A 0.000,B 0.000,C 90.000,E1 336.975} C_DIS
LIN {X -0.035,Y -528.831,Z 720.665,A 0.000,B 0.000,C 90.000,E1 335.665} C_DIS
LIN {X -0.192,Y -535.069,Z 720.663,A 0.000,B 0.000,C 90.000,E1 335.281} C_DIS
LIN {X -0.002,Y -541.099,Z 720.660,A 0.000,B 0.000,C 90.000,E1 334.845} C_DIS
LIN {X -0.172,Y -545.516,Z 720.659,A 0.000,B 0.000,C 90.000,E1 334.537} C_DIS
LIN {X -0.123,Y -553.661,Z 720.655,A 0.000,B 0.000,C 90.000,E1 333.845} C_DIS
LIN {X 0.076,Y -557.794,Z 720.653,A 0.000,B 0.000,C 90.000,E1 333.461} C_DIS
LIN {X -0.308,Y -563.049,Z 720.650,A 0.000,B 0.000,C 90.000,E1 332.999} C_DIS
LIN {X 0.084,Y -569.431,Z 720.646,A 0.000,B 0.000,C 90.000,E1 332.308} C_DIS
LIN {X 0.131,Y -575.725,Z 720.643,A 0.000,B 0.000,C 90.000,E1 331.641} C_DIS
LIN {X -0.135,Y -580.519,Z 720.640,A 0.000,B 0.000,C 90.000,E1 331.129} C_DIS
LIN {X -0.147,Y -590.761,Z 720.633,A 0.000,B 0.000,C 90.000,E1 329.921} C_DIS
LIN {X -0.113,Y -596.395,Z 720.629,A 0.000,B 0.000,C 90.000,E1 329.253} C_DIS
LIN {X -0.149,Y -604.660,Z 720.623,A 0.000,B 0.000,C 90.000,E1 328.201} C_DIS
LIN {X 0.299,Y -610.497,Z 720.619,A 0.000,B 0.000,C 90.000,E1 327.375} C_DIS
LIN {X -0.035,Y -616.063,Z 720.615,A 0.000,B 0.000,C 90.000,E1 326.628} C_DIS
LIN {X -0.320,Y -621.259,Z 720.610,A 0.000,B 0.000,C 90.000,E1 325.881} C_DIS
LIN {X -0.216,Y -626.923,Z 720.605,A 0.000,B 0.000,C 90.000,E1 324.975} C_DIS
LIN {X 0.329,Y -633.005,Z 720.600,A 0.000,B 0.000,C 90.000,E1 323.909} C_DIS
LIN {X 0.064,Y -637.995,Z 720.595,A 0.000,B 0.000,C 90.000,E1 323.050} C_DIS
LIN {X -0.147,Y -642.698,Z 720.590,A 0.000,B 0.000,C 90.000,E1 322.190} C_DIS
LIN {X 0.103,Y -647.887,Z 720.584,A 0.000,B 0.000,C 90.000,E1 321.170} C_DIS
LIN {X -0.082,Y -652.734,Z 720.579,A 0.000,B 0.000,C 90.000,E1 320.194} C_DIS
LIN {X -0.210,Y -657.332,Z 720.573,A 0.000,B 0.000,C 90.000,E1 319.218} C_DIS
LIN {X -0.283,Y -661.651,Z 720.568,A 0.000,B 0.000,C 90.000,E1 318.243} C_DIS
LIN {X 0.133,Y -666.572,Z 720.561,A 0.000,B 0.000,C 90.000,E1 316.986} C_DIS
LIN {X -0.321,Y -670.156,Z 720.556,A 0.000,B 0.000,C 90.000,E1 316.053} C_DIS
LIN {X -0.267,Y -673.562,Z 720.550,A 0.000,B 0.000,C 90.000,E1 315.081} C_DIS
LIN {X -0.167,Y -676.731,Z 720.545,A 0.000,B 0.000,C 90.000,E1 314.109} C_DIS
LIN {X 0.006,Y -680.453,Z 720.538,A 0.000,B 0.000,C 90.000,E1 312.894} C_DIS
LIN {X 0.225,Y -683.236,Z 720.533,A 0.000,B 0.000,C 90.000,E1 311.919} C_DIS
LIN {X -0.077,Y -685.202,Z 720.529,A 0.000,B 0.000,C 90.000,E1 311.229} C_DIS
LIN {X 0.216,Y -687.609,Z 720.524,A 0.000,B 0.000,C 90.000,E1 310.253} C_DIS
LIN {X 0.008,Y -689.798,Z 720.518,A 0.000,B 0.000,C 90.000,E1 309.322} C_DIS
LIN {X -0.080,Y -691.676,Z 720.513,A 0.000,B 0.000,C 90.000,E1 308.382} C_DIS
LIN {X -0.141,Y -693.237,Z 720.508,A 0.000,B 0.000,C 90.000,E1 307.443} C_DIS
LIN {X -0.182,Y -694.621,Z 720.503,A 0.000,B 0.000,C 90.000,E1 306.503} C_DIS
LIN {X 0.004,Y -696.130,Z 720.496,A 0.000,B 0.000,C 90.000,E1 305.311} C_DIS
LIN {X -0.410,Y -697.076,Z 720.491,A 0.000,B 0.000,C 90.000,E1 304.405} C_DIS
LIN {X 0.052,Y -698.364,Z 720.483,A 0.000,B 0.000,C 90.000,E1 302.959} C_DIS
LIN {X 0.163,Y -699.536,Z 720.475,A 0.000,B 0.000,C 90.000,E1 301.544} C_DIS
LIN {X -0.253,Y -700.081,Z 720.471,A 0.000,B 0.000,C 90.000,E1 300.875} C_DIS
LIN {X -0.047,Y -700.544,Z 720.466,A 0.000,B 0.000,C 90.000,E1 299.922} C_DIS
LIN {X 0.076,Y -700.870,Z 720.460,A 0.000,B 0.000,C 90.000,E1 298.743} C_DIS
LIN {X 0.082,Y -701.432,Z 720.449,A 0.000,B 0.000,C 90.000,E1 296.873} C_DIS
LIN {X 0.174,Y -702.103,Z 720.442,A 0.000,B 0.000,C 90.000,E1 295.463} C_DIS
LIN {X 0.152,Y -702.199,Z 720.440,A 0.000,B 0.000,C 90.000,E1 295.232} C_DIS
LIN {X 0.350,Y -701.832,Z 720.436,A 0.000,B 0.000,C 90.000,E1 294.515} C_DIS
LIN {X -0.303,Y -701.102,Z 720.435,A 0.000,B 0.000,C 90.000,E1 294.335} C_DIS
LIN {X 0.243,Y -699.178,Z 720.432,A 0.000,B 0.000,C 90.000,E1 293.823} C_DIS
LIN {X 0.095,Y -698.382,Z 720.432,A 0.000,B 0.000,C 90.000,E1 293.718} C_DIS
LIN {X 0.229,Y -697.199,Z 720.431,A 0.000,B 0.000,C 90.000,E1 293.590} C_DIS
LIN {X -0.384,Y -691.377,Z 720.429,A 0.000,B 0.000,C 90.000,E1 293.206} C_DIS
LIN {X -0.053,Y -689.333,Z 720.428,A 0.000,B 0.000,C 90.000,E1 293.078} C_DIS
LIN {X 0.274,Y -686.527,Z 720.428,A 0.000,B 0.000,C 90.000,E1 292.950} C_DIS
LIN {X -0.018,Y -678.337,Z 720.427,A 0.000,B 0.000,C 90.000,E1 292.770} C_DIS
LIN {X 0.092,Y -675.906,Z 720.426,A 0.000,B 0.000,C 90.000,E1 292.717} C_DIS
LIN {X -0.192,Y -658.136,Z 720.425,A 0.000,B 0.000,C 90.000,E1 292.514} C_DIS
LIN {X -0.006,Y -644.565,Z 720.424,A 0.000,B 0.000,C 90.000,E1 292.280} C_DIS
LIN {X 0.018,Y -634.378,Z 720.423,A 0.000,B 0.000,C 90.000,E1 292.078} C_DIS
LIN {X -0.052,Y -620.958,Z 720.421,A 0.000,B 0.000,C 90.000,E1 291.770} C_DIS
LIN {X 0.091,Y -586.425,Z 720.416,A 0.000,B 0.000,C 90.000,E1 290.791} C_DIS
LIN {X 0.018,Y -574.020,Z 720.414,A 0.000,B 0.000,C 90.000,E1 290.429} C_DIS
LIN {X -0.191,Y -568.539,Z 720.413,A 0.000,B 0.000,C 90.000,E1 290.301} C_DIS
LIN {X 0.339,Y -561.221,Z 720.411,A 0.000,B 0.000,C 90.000,E1 289.993} C_DIS
LIN {X 0.264,Y -559.910,Z 720.411,A 0.000,B 0.000,C 90.000,E1 289.939} C_DIS
LIN {X -0.185,Y -556.434,Z 720.410,A 0.000,B 0.000,C 90.000,E1 289.758} C_DIS
LIN {X -0.243,Y -556.347,Z 720.410,A 0.000,B 0.000,C 90.000,E1 289.758} C_DIS
LIN {X -0.173,Y -555.480,Z 720.409,A 0.000,B 0.000,C 90.000,E1 289.577} C_DIS
LIN {X -0.003,Y -554.800,Z 720.406,A 0.000,B 0.000,C 90.000,E1 289.141} C_DIS
LIN {X -0.156,Y -554.412,Z 720.400,A 0.000,B 0.000,C 90.000,E1 288.055} C_DIS
LIN {X 0.055,Y -553.638,Z 720.389,A 0.000,B 0.000,C 90.000,E1 286.079} C_DIS
LIN {X 0.093,Y -552.951,Z 720.379,A 0.000,B 0.000,C 90.000,E1 284.120} C_DIS
LIN {X -0.026,Y -552.342,Z 720.368,A 0.000,B 0.000,C 90.000,E1 282.175} C_DIS
LIN {X 0.153,Y -551.536,Z 720.357,A 0.000,B 0.000,C 90.000,E1 280.197} C_DIS
LIN {X 0.094,Y -550.887,Z 720.349,A 0.000,B 0.000,C 90.000,E1 278.803} C_DIS
LIN {X 0.153,Y -549.955,Z 720.338,A 0.000,B 0.000,C 90.000,E1 276.834} C_DIS
LIN {X 0.200,Y -549.162,Z 720.324,A 0.000,B 0.000,C 90.000,E1 274.302} C_DIS
LIN {X -0.044,Y -548.674,Z 720.316,A 0.000,B 0.000,C 90.000,E1 272.922} C_DIS
LIN {X 0.265,Y -547.993,Z 720.307,A 0.000,B 0.000,C 90.000,E1 271.203} C_DIS
LIN {X -0.091,Y -547.414,Z 720.301,A 0.000,B 0.000,C 90.000,E1 270.115} C_DIS
LIN {X 0.179,Y -546.413,Z 720.291,A 0.000,B 0.000,C 90.000,E1 268.396} C_DIS
LIN {X -0.084,Y -545.329,Z 720.282,A 0.000,B 0.000,C 90.000,E1 266.731} C_DIS
LIN {X 0.113,Y -544.346,Z 720.274,A 0.000,B 0.000,C 90.000,E1 265.298} C_DIS
LIN {X -0.070,Y -542.897,Z 720.263,A 0.000,B 0.000,C 90.000,E1 263.337} C_DIS
LIN {X 0.251,Y -541.424,Z 720.254,A 0.000,B 0.000,C 90.000,E1 261.602} C_DIS
LIN {X 0.013,Y -540.233,Z 720.246,A 0.000,B 0.000,C 90.000,E1 260.208} C_DIS
LIN {X -0.111,Y -538.479,Z 720.235,A 0.000,B 0.000,C 90.000,E1 258.229} C_DIS
LIN {X -0.123,Y -537.004,Z 720.225,A 0.000,B 0.000,C 90.000,E1 256.520} C_DIS
LIN {X 0.055,Y -536.214,Z 720.220,A 0.000,B 0.000,C 90.000,E1 255.644} C_DIS
LIN {X 0.121,Y -534.422,Z 720.211,A 0.000,B 0.000,C 90.000,E1 253.921} C_DIS
LIN {X 0.075,Y -533.282,Z 720.204,A 0.000,B 0.000,C 90.000,E1 252.779} C_DIS
LIN {X 0.208,Y -531.830,Z 720.196,A 0.000,B 0.000,C 90.000,E1 251.329} C_DIS
LIN {X -0.067,Y -530.784,Z 720.192,A 0.000,B 0.000,C 90.000,E1 250.496} C_DIS
LIN {X -0.123,Y -528.551,Z 720.182,A 0.000,B 0.000,C 90.000,E1 248.773} C_DIS
LIN {X -0.087,Y -526.900,Z 720.176,A 0.000,B 0.000,C 90.000,E1 247.614} C_DIS
LIN {X -0.196,Y -524.744,Z 720.168,A 0.000,B 0.000,C 90.000,E1 246.177} C_DIS
LIN {X -0.123,Y -522.362,Z 720.159,A 0.000,B 0.000,C 90.000,E1 244.717} C_DIS
LIN {X -0.092,Y -519.957,Z 720.151,A 0.000,B 0.000,C 90.000,E1 243.256} C_DIS
LIN {X -0.244,Y -517.709,Z 720.145,A 0.000,B 0.000,C 90.000,E1 242.103} C_DIS
LIN {X -0.170,Y -514.212,Z 720.135,A 0.000,B 0.000,C 90.000,E1 240.333} C_DIS
LIN {X 0.187,Y -512.414,Z 720.130,A 0.000,B 0.000,C 90.000,E1 239.410} C_DIS
LIN {X -0.042,Y -508.717,Z 720.120,A 0.000,B 0.000,C 90.000,E1 237.661} C_DIS
LIN {X -0.077,Y -505.022,Z 720.110,A 0.000,B 0.000,C 90.000,E1 235.881} C_DIS
LIN {X -0.209,Y -501.629,Z 720.102,A 0.000,B 0.000,C 90.000,E1 234.402} C_DIS
LIN {X -0.279,Y -498.742,Z 720.095,A 0.000,B 0.000,C 90.000,E1 233.210} C_DIS
LIN {X 0.193,Y -491.812,Z 720.080,A 0.000,B 0.000,C 90.000,E1 230.436} C_DIS
LIN {X 0.017,Y -486.817,Z 720.069,A 0.000,B 0.000,C 90.000,E1 228.324} C_DIS
LIN {X -0.055,Y -484.020,Z 720.062,A 0.000,B 0.000,C 90.000,E1 227.106} C_DIS
LIN {X 0.069,Y -479.882,Z 720.051,A 0.000,B 0.000,C 90.000,E1 225.243} C_DIS
LIN {X -0.116,Y -475.219,Z 720.039,A 0.000,B 0.000,C 90.000,E1 223.095} C_DIS
LIN {X -0.166,Y -471.289,Z 720.029,A 0.000,B 0.000,C 90.000,E1 221.229} C_DIS
LIN {X -0.031,Y -467.897,Z 720.020,A 0.000,B 0.000,C 90.000,E1 219.644} C_DIS
LIN {X -0.021,Y -465.128,Z 720.013,A 0.000,B 0.000,C 90.000,E1 218.382} C_DIS
LIN {X 0.051,Y -458.805,Z 719.997,A 0.000,B 0.000,C 90.000,E1 215.518} C_DIS
LIN {X 0.212,Y -455.161,Z 719.987,A 0.000,B 0.000,C 90.000,E1 213.579} C_DIS
LIN {X -0.052,Y -452.128,Z 719.978,A 0.000,B 0.000,C 90.000,E1 212.005} C_DIS
LIN {X 0.002,Y -449.201,Z 719.969,A 0.000,B 0.000,C 90.000,E1 210.384} C_DIS
LIN {X 0.156,Y -446.137,Z 719.960,A 0.000,B 0.000,C 90.000,E1 208.743} C_DIS
LIN {X 0.041,Y -443.249,Z 719.951,A 0.000,B 0.000,C 90.000,E1 207.129} C_DIS
LIN {X -0.170,Y -440.827,Z 719.944,A 0.000,B 0.000,C 90.000,E1 205.848} C_DIS
LIN {X -0.183,Y -437.854,Z 719.934,A 0.000,B 0.000,C 90.000,E1 204.207} C_DIS
LIN {X -0.031,Y -434.157,Z 719.923,A 0.000,B 0.000,C 90.000,E1 202.206} C_DIS
LIN {X -0.108,Y -431.061,Z 719.914,A 0.000,B 0.000,C 90.000,E1 200.556} C_DIS
LIN {X -0.032,Y -427.478,Z 719.903,A 0.000,B 0.000,C 90.000,E1 198.544} C_DIS
LIN {X 0.025,Y -424.340,Z 719.894,A 0.000,B 0.000,C 90.000,E1 196.858} C_DIS
LIN {X -0.101,Y -421.194,Z 719.884,A 0.000,B 0.000,C 90.000,E1 195.190} C_DIS
LIN {X 0.012,Y -418.193,Z 719.875,A 0.000,B 0.000,C 90.000,E1 193.480} C_DIS
LIN {X 0.113,Y -414.593,Z 719.864,A 0.000,B 0.000,C 90.000,E1 191.422} C_DIS
LIN {X 0.064,Y -410.367,Z 719.850,A 0.000,B 0.000,C 90.000,E1 189.029} C_DIS
LIN {X 0.114,Y -406.604,Z 719.837,A 0.000,B 0.000,C 90.000,E1 186.606} C_DIS
LIN {X 0.065,Y -403.500,Z 719.825,A 0.000,B 0.000,C 90.000,E1 184.531} C_DIS
LIN {X -0.124,Y -400.583,Z 719.814,A 0.000,B 0.000,C 90.000,E1 182.465} C_DIS
LIN {X -0.050,Y -397.646,Z 719.800,A 0.000,B 0.000,C 90.000,E1 180.000} C_DIS
LIN {X -0.171,Y -394.490,Z 719.782,A 0.000,B 0.000,C 90.000,E1 176.846} C_DIS
LIN {X 0.083,Y -392.263,Z 719.767,A 0.000,B 0.000,C 90.000,E1 173.976} C_DIS
LIN {X 0.033,Y -390.530,Z 719.751,A 0.000,B 0.000,C 90.000,E1 171.141} C_DIS
LIN {X 0.104,Y -389.645,Z 719.739,A 0.000,B 0.000,C 90.000,E1 168.993} C_DIS
LIN {X -0.047,Y -389.171,Z 719.731,A 0.000,B 0.000,C 90.000,E1 167.589} C_DIS
LIN {X -0.194,Y -388.369,Z 719.715,A 0.000,B 0.000,C 90.000,E1 164.755} C_DIS
LIN {X -0.043,Y -387.933,Z 719.699,A 0.000,B 0.000,C 90.000,E1 161.873} C_DIS
LIN {X -0.181,Y -387.703,Z 719.685,A 0.000,B 0.000,C 90.000,E1 159.390} C_DIS
LIN {X 0.109,Y -387.652,Z 719.669,A 0.000,B 0.000,C 90.000,E1 156.485} C_DIS
LIN {X 0.156,Y -387.764,Z 719.658,A 0.000,B 0.000,C 90.000,E1 154.332} C_DIS
LIN {X -0.145,Y -388.044,Z 719.646,A 0.000,B 0.000,C 90.000,E1 152.231} C_DIS
LIN {X 0.073,Y -388.431,Z 719.636,A 0.000,B 0.000,C 90.000,E1 150.411} C_DIS
LIN {X 0.027,Y -390.441,Z 719.612,A 0.000,B 0.000,C 90.000,E1 146.135} C_DIS
LIN {X -0.102,Y -394.937,Z 719.586,A 0.000,B 0.000,C 90.000,E1 141.537} C_DIS
LIN {X 0.168,Y -397.822,Z 719.575,A 0.000,B 0.000,C 90.000,E1 139.380} C_DIS
LIN {X -0.012,Y -400.396,Z 719.567,A 0.000,B 0.000,C 90.000,E1 138.000} C_DIS
LIN {X -0.089,Y -402.269,Z 719.563,A 0.000,B 0.000,C 90.000,E1 137.310} C_DIS
LIN {X -0.062,Y -404.406,Z 719.560,A 0.000,B 0.000,C 90.000,E1 136.782} C_DIS
LIN {X -0.013,Y -407.396,Z 719.557,A 0.000,B 0.000,C 90.000,E1 136.257} C_DIS
LIN {X -0.022,Y -411.508,Z 719.554,A 0.000,B 0.000,C 90.000,E1 135.729} C_DIS
LIN {X 0.119,Y -419.603,Z 719.549,A 0.000,B 0.000,C 90.000,E1 134.838} C_DIS
LIN {X 0.232,Y -441.975,Z 719.537,A 0.000,B 0.000,C 90.000,E1 132.690} C_DIS
LIN {X -0.162,Y -447.936,Z 719.534,A 0.000,B 0.000,C 90.000,E1 132.204} C_DIS
LIN {X -0.201,Y -461.392,Z 719.528,A 0.000,B 0.000,C 90.000,E1 130.987} C_DIS
LIN {X -0.219,Y -470.109,Z 719.523,A 0.000,B 0.000,C 90.000,E1 130.172} C_DIS
LIN {X -0.212,Y -477.219,Z 719.519,A 0.000,B 0.000,C 90.000,E1 129.483} C_DIS
LIN {X 0.034,Y -484.215,Z 719.515,A 0.000,B 0.000,C 90.000,E1 128.749} C_DIS
LIN {X 0.053,Y -490.893,Z 719.511,A 0.000,B 0.000,C 90.000,E1 128.051} C_DIS
LIN {X -0.152,Y -496.034,Z 719.508,A 0.000,B 0.000,C 90.000,E1 127.523} C_DIS
LIN {X -0.229,Y -501.253,Z 719.505,A 0.000,B 0.000,C 90.000,E1 126.950} C_DIS
LIN {X 0.161,Y -505.075,Z 719.503,A 0.000,B 0.000,C 90.000,E1 126.457} C_DIS
LIN {X 0.172,Y -509.625,Z 719.500,A 0.000,B 0.000,C 90.000,E1 125.884} C_DIS
LIN {X 0.048,Y -513.923,Z 719.496,A 0.000,B 0.000,C 90.000,E1 125.311} C_DIS
LIN {X 0.058,Y -517.743,Z 719.493,A 0.000,B 0.000,C 90.000,E1 124.771} C_DIS
LIN {X -0.068,Y -521.522,Z 719.490,A 0.000,B 0.000,C 90.000,E1 124.199} C_DIS
LIN {X 0.098,Y -525.764,Z 719.486,A 0.000,B 0.000,C 90.000,E1 123.452} C_DIS
LIN {X -0.135,Y -529.662,Z 719.482,A 0.000,B 0.000,C 90.000,E1 122.752} C_DIS
LIN {X 0.262,Y -532.654,Z 719.479,A 0.000,B 0.000,C 90.000,E1 122.133} C_DIS
LIN {X 0.245,Y -537.149,Z 719.473,A 0.000,B 0.000,C 90.000,E1 121.131} C_DIS
LIN {X 0.152,Y -542.056,Z 719.467,A 0.000,B 0.000,C 90.000,E1 120.001} C_DIS
LIN {X -0.134,Y -547.758,Z 719.459,A 0.000,B 0.000,C 90.000,E1 118.615} C_DIS
LIN {X -0.121,Y -550.960,Z 719.454,A 0.000,B 0.000,C 90.000,E1 117.769} C_DIS
LIN {X 0.193,Y -554.913,Z 719.448,A 0.000,B 0.000,C 90.000,E1 116.616} C_DIS
LIN {X -0.177,Y -558.391,Z 719.442,A 0.000,B 0.000,C 90.000,E1 115.540} C_DIS
LIN {X -0.061,Y -560.655,Z 719.437,A 0.000,B 0.000,C 90.000,E1 114.695} C_DIS
LIN {X 0.352,Y -562.621,Z 719.433,A 0.000,B 0.000,C 90.000,E1 113.823} C_DIS
LIN {X 0.052,Y -564.358,Z 719.428,A 0.000,B 0.000,C 90.000,E1 113.025} C_DIS
LIN {X -0.010,Y -565.836,Z 719.423,A 0.000,B 0.000,C 90.000,E1 112.206} C_DIS
LIN {X -0.131,Y -568.113,Z 719.416,A 0.000,B 0.000,C 90.000,E1 110.844} C_DIS
LIN {X 0.088,Y -571.116,Z 719.405,A 0.000,B 0.000,C 90.000,E1 108.906} C_DIS
LIN {X 0.044,Y -572.739,Z 719.399,A 0.000,B 0.000,C 90.000,E1 107.819} C_DIS
LIN {X 0.207,Y -574.626,Z 719.391,A 0.000,B 0.000,C 90.000,E1 106.441} C_DIS
LIN {X -0.308,Y -576.503,Z 719.384,A 0.000,B 0.000,C 90.000,E1 105.134} C_DIS
LIN {X 0.114,Y -577.980,Z 719.378,A 0.000,B 0.000,C 90.000,E1 104.008} C_DIS
LIN {X 0.086,Y -580.445,Z 719.367,A 0.000,B 0.000,C 90.000,E1 102.119} C_DIS
LIN {X -0.024,Y -582.284,Z 719.360,A 0.000,B 0.000,C 90.000,E1 100.782} C_DIS
LIN {X -0.093,Y -583.989,Z 719.352,A 0.000,B 0.000,C 90.000,E1 99.443} C_DIS
LIN {X 0.200,Y -585.245,Z 719.346,A 0.000,B 0.000,C 90.000,E1 98.341} C_DIS
LIN {X -0.004,Y -587.256,Z 719.336,A 0.000,B 0.000,C 90.000,E1 96.486} C_DIS
LIN {X -0.150,Y -588.605,Z 719.329,A 0.000,B 0.000,C 90.000,E1 95.163} C_DIS
LIN {X 0.079,Y -589.710,Z 719.323,A 0.000,B 0.000,C 90.000,E1 94.073} C_DIS
LIN {X -0.226,Y -590.705,Z 719.317,A 0.000,B 0.000,C 90.000,E1 93.037} C_DIS
LIN {X -0.145,Y -591.967,Z 719.308,A 0.000,B 0.000,C 90.000,E1 91.432} C_DIS
LIN {X -0.263,Y -592.810,Z 719.301,A 0.000,B 0.000,C 90.000,E1 90.115} C_DIS
LIN {X 0.228,Y -593.473,Z 719.293,A 0.000,B 0.000,C 90.000,E1 88.740} C_DIS
LIN {X -0.226,Y -594.043,Z 719.284,A 0.000,B 0.000,C 90.000,E1 87.192} C_DIS
LIN {X -0.258,Y -594.308,Z 719.277,A 0.000,B 0.000,C 90.000,E1 85.869} C_DIS
LIN {X -0.067,Y -594.502,Z 719.268,A 0.000,B 0.000,C 90.000,E1 84.261} C_DIS
LIN {X -0.024,Y -594.502,Z 719.261,A 0.000,B 0.000,C 90.000,E1 82.932} C_DIS
LIN {X -0.255,Y -594.380,Z 719.255,A 0.000,B 0.000,C 90.000,E1 81.894} C_DIS
LIN {X -0.126,Y -594.057,Z 719.247,A 0.000,B 0.000,C 90.000,E1 80.557} C_DIS
LIN {X 0.002,Y -593.479,Z 719.240,A 0.000,B 0.000,C 90.000,E1 79.218} C_DIS
LIN {X -0.196,Y -592.494,Z 719.231,A 0.000,B 0.000,C 90.000,E1 77.645} C_DIS
LIN {X -0.159,Y -591.413,Z 719.222,A 0.000,B 0.000,C 90.000,E1 76.047} C_DIS
LIN {X -0.136,Y -590.116,Z 719.214,A 0.000,B 0.000,C 90.000,E1 74.448} C_DIS
LIN {X 0.160,Y -588.938,Z 719.206,A 0.000,B 0.000,C 90.000,E1 73.087} C_DIS
LIN {X 0.036,Y -587.598,Z 719.199,A 0.000,B 0.000,C 90.000,E1 71.764} C_DIS
LIN {X -0.257,Y -585.798,Z 719.190,A 0.000,B 0.000,C 90.000,E1 70.188} C_DIS
LIN {X 0.096,Y -584.495,Z 719.184,A 0.000,B 0.000,C 90.000,E1 69.082} C_DIS
LIN {X 0.077,Y -582.645,Z 719.176,A 0.000,B 0.000,C 90.000,E1 67.741} C_DIS
LIN {X -0.068,Y -580.546,Z 719.169,A 0.000,B 0.000,C 90.000,E1 66.410} C_DIS
LIN {X -0.331,Y -578.536,Z 719.163,A 0.000,B 0.000,C 90.000,E1 65.357} C_DIS
LIN {X -0.238,Y -576.910,Z 719.158,A 0.000,B 0.000,C 90.000,E1 64.537} C_DIS
LIN {X -0.062,Y -574.499,Z 719.152,A 0.000,B 0.000,C 90.000,E1 63.435} C_DIS
LIN {X -0.177,Y -571.731,Z 719.146,A 0.000,B 0.000,C 90.000,E1 62.359} C_DIS
LIN {X 0.267,Y -570.326,Z 719.143,A 0.000,B 0.000,C 90.000,E1 61.769} C_DIS
LIN {X -0.147,Y -567.091,Z 719.137,A 0.000,B 0.000,C 90.000,E1 60.717} C_DIS
LIN {X -0.117,Y -563.413,Z 719.131,A 0.000,B 0.000,C 90.000,E1 59.616} C_DIS
LIN {X -0.135,Y -560.454,Z 719.127,A 0.000,B 0.000,C 90.000,E1 58.791} C_DIS
LIN {X 0.219,Y -558.305,Z 719.124,A 0.000,B 0.000,C 90.000,E1 58.201} C_DIS
LIN {X -0.033,Y -555.381,Z 719.120,A 0.000,B 0.000,C 90.000,E1 57.533} C_DIS
LIN {X -0.013,Y -552.200,Z 719.116,A 0.000,B 0.000,C 90.000,E1 56.834} C_DIS
LIN {X -0.018,Y -548.547,Z 719.112,A 0.000,B 0.000,C 90.000,E1 56.135} C_DIS
LIN {X -0.207,Y -542.908,Z 719.107,A 0.000,B 0.000,C 90.000,E1 55.182} C_DIS
LIN {X -0.005,Y -540.283,Z 719.104,A 0.000,B 0.000,C 90.000,E1 54.736} C_DIS
LIN {X -0.127,Y -537.571,Z 719.102,A 0.000,B 0.000,C 90.000,E1 54.322} C_DIS
LIN {X -0.103,Y -533.546,Z 719.099,A 0.000,B 0.000,C 90.000,E1 53.749} C_DIS
LIN {X 0.316,Y -529.081,Z 719.095,A 0.000,B 0.000,C 90.000,E1 53.130} C_DIS
LIN {X -0.130,Y -524.416,Z 719.092,A 0.000,B 0.000,C 90.000,E1 52.637} C_DIS
LIN {X -0.199,Y -519.316,Z 719.089,A 0.000,B 0.000,C 90.000,E1 52.110} C_DIS
LIN {X -0.138,Y -515.002,Z 719.087,A 0.000,B 0.000,C 90.000,E1 51.698} C_DIS
LIN {X 0.102,Y -508.894,Z 719.084,A 0.000,B 0.000,C 90.000,E1 51.170} C_DIS
LIN {X 0.186,Y -504.235,Z 719.082,A 0.000,B 0.000,C 90.000,E1 50.803} C_DIS
LIN {X 0.007,Y -499.451,Z 719.081,A 0.000,B 0.000,C 90.000,E1 50.481} C_DIS
LIN {X 0.278,Y -491.319,Z 719.078,A 0.000,B 0.000,C 90.000,E1 49.908} C_DIS
LIN {X -0.075,Y -484.676,Z 719.075,A 0.000,B 0.000,C 90.000,E1 49.542} C_DIS
LIN {X 0.125,Y -468.245,Z 719.070,A 0.000,B 0.000,C 90.000,E1 48.528} C_DIS
LIN {X -0.198,Y -450.414,Z 719.064,A 0.000,B 0.000,C 90.000,E1 47.472} C_DIS
LIN {X 0.003,Y -426.449,Z 719.055,A 0.000,B 0.000,C 90.000,E1 45.850} C_DIS
LIN {X -0.131,Y -420.280,Z 719.052,A 0.000,B 0.000,C 90.000,E1 45.405} C_DIS
LIN {X -0.006,Y -419.544,Z 719.052,A 0.000,B 0.000,C 90.000,E1 45.324} C_DIS
LIN {X -0.034,Y -419.510,Z 719.052,A 0.000,B 0.000,C 90.000,E1 45.324} C_DIS
LIN {X -0.038,Y -418.578,Z 719.049,A 0.000,B 0.000,C 90.000,E1 44.798} C_DIS
LIN {X 0.078,Y -409.015,Z 719.024,A 0.000,B 0.000,C 90.000,E1 40.334} C_DIS
LIN {X 0.058,Y -406.690,Z 719.017,A 0.000,B 0.000,C 90.000,E1 38.955} C_DIS
LIN {X -0.052,Y -407.210,Z 718.996,A 0.000,B 0.000,C 90.000,E1 35.311} C_DIS
LIN {X 0.007,Y -408.149,Z 718.983,A 0.000,B 0.000,C 90.000,E1 32.880} C_DIS
LIN {X 0.074,Y -409.078,Z 718.971,A 0.000,B 0.000,C 90.000,E1 30.797} C_DIS
LIN {X -0.045,Y -410.203,Z 718.960,A 0.000,B 0.000,C 90.000,E1 28.743} C_DIS
LIN {X 0.019,Y -411.422,Z 718.948,A 0.000,B 0.000,C 90.000,E1 26.668} C_DIS
LIN {X 0.082,Y -413.661,Z 718.931,A 0.000,B 0.000,C 90.000,E1 23.567} C_DIS
LIN {X -0.083,Y -415.463,Z 718.920,A 0.000,B 0.000,C 90.000,E1 21.535} C_DIS
LIN {X 0.034,Y -417.168,Z 718.910,A 0.000,B 0.000,C 90.000,E1 19.812} C_DIS
LIN {X 0.003,Y -420.232,Z 718.895,A 0.000,B 0.000,C 90.000,E1 17.094} C_DIS
LIN {X 0.054,Y -423.301,Z 718.882,A 0.000,B 0.000,C 90.000,E1 14.717} C_DIS
LIN {X -0.002,Y -426.042,Z 718.871,A 0.000,B 0.000,C 90.000,E1 12.703} C_DIS
LIN {X -0.088,Y -429.356,Z 718.858,A 0.000,B 0.000,C 90.000,E1 10.366} C_DIS
LIN {X 0.200,Y -432.702,Z 718.845,A 0.000,B 0.000,C 90.000,E1 7.992} C_DIS
LIN {X 0.230,Y -436.621,Z 718.830,A 0.000,B 0.000,C 90.000,E1 5.334} C_DIS
LIN {X 0.048,Y -441.952,Z 718.812,A 0.000,B 0.000,C 90.000,E1 2.064} C_DIS
LIN {X 0.169,Y -445.994,Z 718.799,A 0.000,B 0.000,C 90.000,E1 359.771} C_DIS
LIN {X 0.007,Y -449.172,Z 718.790,A 0.000,B 0.000,C 90.000,E1 358.165} C_DIS
LIN {X -0.028,Y -454.261,Z 718.776,A 0.000,B 0.000,C 90.000,E1 355.584} C_DIS
LIN {X 0.209,Y -458.372,Z 718.765,A 0.000,B 0.000,C 90.000,E1 353.628} C_DIS
LIN {X -0.050,Y -461.686,Z 718.756,A 0.000,B 0.000,C 90.000,E1 352.064} C_DIS
LIN {X 0.218,Y -464.928,Z 718.747,A 0.000,B 0.000,C 90.000,E1 350.443} C_DIS
LIN {X -0.105,Y -467.383,Z 718.740,A 0.000,B 0.000,C 90.000,E1 349.218} C_DIS
LIN {X -0.118,Y -470.375,Z 718.731,A 0.000,B 0.000,C 90.000,E1 347.645} C_DIS
LIN {X -0.213,Y -474.340,Z 718.719,A 0.000,B 0.000,C 90.000,E1 345.463} C_DIS
LIN {X -0.141,Y -476.077,Z 718.714,A 0.000,B 0.000,C 90.000,E1 344.519} C_DIS
LIN {X 0.139,Y -481.474,Z 718.698,A 0.000,B 0.000,C 90.000,E1 341.692} C_DIS
LIN {X -0.185,Y -484.820,Z 718.690,A 0.000,B 0.000,C 90.000,E1 340.188} C_DIS
LIN {X -0.169,Y -486.466,Z 718.686,A 0.000,B 0.000,C 90.000,E1 339.571} C_DIS
LIN {X -0.155,Y -487.397,Z 718.685,A 0.000,B 0.000,C 90.000,E1 339.263} C_DIS
LIN {X 0.101,Y -489.185,Z 718.682,A 0.000,B 0.000,C 90.000,E1 338.773} C_DIS
LIN {X 0.127,Y -490.687,Z 718.680,A 0.000,B 0.000,C 90.000,E1 338.465} C_DIS
LIN {X 0.222,Y -492.988,Z 718.679,A 0.000,B 0.000,C 90.000,E1 338.103} C_DIS
LIN {X 0.109,Y -496.966,Z 718.676,A 0.000,B 0.000,C 90.000,E1 337.667} C_DIS
LIN {X 0.064,Y -502.069,Z 718.674,A 0.000,B 0.000,C 90.000,E1 337.230} C_DIS
LIN {X 0.196,Y -508.385,Z 718.671,A 0.000,B 0.000,C 90.000,E1 336.741} C_DIS
LIN {X 0.214,Y -527.700,Z 718.664,A 0.000,B 0.000,C 90.000,E1 335.485} C_DIS
LIN {X 0.257,Y -535.575,Z 718.661,A 0.000,B 0.000,C 90.000,E1 334.973} C_DIS
LIN {X -0.064,Y -541.521,Z 718.659,A 0.000,B 0.000,C 90.000,E1 334.588} C_DIS
LIN {X -0.292,Y -545.954,Z 718.657,A 0.000,B 0.000,C 90.000,E1 334.280} C_DIS
LIN {X 0.223,Y -552.972,Z 718.654,A 0.000,B 0.000,C 90.000,E1 333.640} C_DIS
LIN {X -0.024,Y -559.871,Z 718.650,A 0.000,B 0.000,C 90.000,E1 333.050} C_DIS
LIN {X -0.044,Y -566.411,Z 718.647,A 0.000,B 0.000,C 90.000,E1 332.410} C_DIS
LIN {X -0.293,Y -574.002,Z 718.642,A 0.000,B 0.000,C 90.000,E1 331.641} C_DIS
LIN {X 0.232,Y -580.017,Z 718.639,A 0.000,B 0.000,C 90.000,E1 330.923} C_DIS
LIN {X -0.051,Y -590.386,Z 718.632,A 0.000,B 0.000,C 90.000,E1 329.744} C_DIS
LIN {X -0.023,Y -595.960,Z 718.628,A 0.000,B 0.000,C 90.000,E1 329.076} C_DIS
LIN {X 0.286,Y -603.329,Z 718.623,A 0.000,B 0.000,C 90.000,E1 328.122} C_DIS
LIN {X -0.082,Y -608.300,Z 718.619,A 0.000,B 0.000,C 90.000,E1 327.502} C_DIS
LIN {X 0.075,Y -614.003,Z 718.615,A 0.000,B 0.000,C 90.000,E1 326.707} C_DIS
LIN {X -0.212,Y -618.462,Z 718.612,A 0.000,B 0.000,C 90.000,E1 326.087} C_DIS
LIN {X -0.138,Y -624.328,Z 718.607,A 0.000,B 0.000,C 90.000,E1 325.182} C_DIS
LIN {X 0.071,Y -629.820,Z 718.602,A 0.000,B 0.000,C 90.000,E1 324.276} C_DIS
LIN {X -0.234,Y -635.046,Z 718.597,A 0.000,B 0.000,C 90.000,E1 323.417} C_DIS
LIN {X -0.089,Y -640.578,Z 718.591,A 0.000,B 0.000,C 90.000,E1 322.396} C_DIS
LIN {X 0.135,Y -645.862,Z 718.586,A 0.000,B 0.000,C 90.000,E1 321.376} C_DIS
LIN {X -0.061,Y -651.492,Z 718.579,A 0.000,B 0.000,C 90.000,E1 320.275} C_DIS
LIN {X -0.204,Y -656.176,Z 718.574,A 0.000,B 0.000,C 90.000,E1 319.299} C_DIS
LIN {X -0.319,Y -661.629,Z 718.567,A 0.000,B 0.000,C 90.000,E1 318.081} C_DIS
LIN {X 0.116,Y -664.664,Z 718.563,A 0.000,B 0.000,C 90.000,E1 317.310} C_DIS
LIN {X 0.097,Y -667.551,Z 718.559,A 0.000,B 0.000,C 90.000,E1 316.581} C_DIS
LIN {X -0.333,Y -671.995,Z 718.552,A 0.000,B 0.000,C 90.000,E1 315.405} C_DIS
LIN {X -0.253,Y -675.281,Z 718.547,A 0.000,B 0.000,C 90.000,E1 314.433} C_DIS
LIN {X -0.100,Y -679.114,Z 718.540,A 0.000,B 0.000,C 90.000,E1 313.218} C_DIS
LIN {X 0.102,Y -682.025,Z 718.535,A 0.000,B 0.000,C 90.000,E1 312.243} C_DIS
LIN {X -0.158,Y -684.724,Z 718.529,A 0.000,B 0.000,C 90.000,E1 311.310} C_DIS
LIN {X 0.130,Y -687.238,Z 718.524,A 0.000,B 0.000,C 90.000,E1 310.334} C_DIS
LIN {X -0.139,Y -688.935,Z 718.520,A 0.000,B 0.000,C 90.000,E1 309.644} C_DIS
LIN {X 0.138,Y -690.485,Z 718.516,A 0.000,B 0.000,C 90.000,E1 308.910} C_DIS
LIN {X -0.112,Y -691.866,Z 718.512,A 0.000,B 0.000,C 90.000,E1 308.222} C_DIS
LIN {X -0.174,Y -693.433,Z 718.507,A 0.000,B 0.000,C 90.000,E1 307.282} C_DIS
LIN {X 0.342,Y -694.814,Z 718.502,A 0.000,B 0.000,C 90.000,E1 306.297} C_DIS
LIN {X -0.035,Y -696.330,Z 718.495,A 0.000,B 0.000,C 90.000,E1 305.152} C_DIS
LIN {X 0.124,Y -697.276,Z 718.490,A 0.000,B 0.000,C 90.000,E1 304.199} C_DIS
LIN {X -0.034,Y -698.385,Z 718.484,A 0.000,B 0.000,C 90.000,E1 303.038} C_DIS
LIN {X 0.083,Y -699.552,Z 718.476,A 0.000,B 0.000,C 90.000,E1 301.623} C_DIS
LIN {X 0.292,Y -700.263,Z 718.471,A 0.000,B 0.000,C 90.000,E1 300.669} C_DIS
LIN {X 0.148,Y -700.697,Z 718.465,A 0.000,B 0.000,C 90.000,E1 299.745} C_DIS
LIN {X -0.059,Y -701.070,Z 718.458,A 0.000,B 0.000,C 90.000,E1 298.359} C_DIS
LIN {X -0.045,Y -701.711,Z 718.447,A 0.000,B 0.000,C 90.000,E1 296.488} C_DIS
LIN {X 0.128,Y -702.186,Z 718.442,A 0.000,B 0.000,C 90.000,E1 295.540} C_DIS
LIN {X 0.050,Y -702.294,Z 718.439,A 0.000,B 0.000,C 90.000,E1 295.079} C_DIS
LIN {X -0.327,Y -701.947,Z 718.437,A 0.000,B 0.000,C 90.000,E1 294.643} C_DIS
LIN {X -0.051,Y -701.408,Z 718.435,A 0.000,B 0.000,C 90.000,E1 294.387} C_DIS
LIN {X 0.210,Y -699.486,Z 718.433,A 0.000,B 0.000,C 90.000,E1 293.898} C_DIS
LIN {X -0.294,Y -698.870,Z 718.432,A 0.000,B 0.000,C 90.000,E1 293.823} C_DIS
LIN {X -0.160,Y -697.941,Z 718.432,A 0.000,B 0.000,C 90.000,E1 293.695} C_DIS
LIN {X -0.029,Y -696.561,Z 718.431,A 0.000,B 0.000,C 90.000,E1 293.567} C_DIS
LIN {X -0.148,Y -692.211,Z 718.429,A 0.000,B 0.000,C 90.000,E1 293.259} C_DIS
LIN {X 0.186,Y -690.614,Z 718.429,A 0.000,B 0.000,C 90.000,E1 293.131} C_DIS
LIN {X 0.247,Y -688.183,Z 718.428,A 0.000,B 0.000,C 90.000,E1 293.025} C_DIS
LIN {X 0.330,Y -686.252,Z 718.428,A 0.000,B 0.000,C 90.000,E1 292.950} C_DIS
LIN {X 0.127,Y -677.943,Z 718.427,A 0.000,B 0.000,C 90.000,E1 292.770} C_DIS
LIN {X -0.161,Y -670.783,Z 718.426,A 0.000,B 0.000,C 90.000,E1 292.695} C_DIS
LIN {X 0.324,Y -659.820,Z 718.425,A 0.000,B 0.000,C 90.000,E1 292.514} C_DIS
LIN {X -0.036,Y -646.214,Z 718.424,A 0.000,B 0.000,C 90.000,E1 292.333} C_DIS
LIN {X -0.128,Y -636.353,Z 718.423,A 0.000,B 0.000,C 90.000,E1 292.153} C_DIS
LIN {X -0.117,Y -622.898,Z 718.421,A 0.000,B 0.000,C 90.000,E1 291.844} C_DIS
LIN {X 0.062,Y -598.797,Z 718.418,A 0.000,B 0.000,C 90.000,E1 291.173} C_DIS
LIN {X 0.253,Y -574.270,Z 718.414,A 0.000,B 0.000,C 90.000,E1 290.429} C_DIS
LIN {X 0.031,Y -568.791,Z 718.413,A 0.000,B 0.000,C 90.000,E1 290.301} C_DIS
LIN {X -0.255,Y -561.232,Z 718.411,A 0.000,B 0.000,C 90.000,E1 290.066} C_DIS
LIN {X 0.129,Y -559.476,Z 718.411,A 0.000,B 0.000,C 90.000,E1 289.939} C_DIS
LIN {X -0.080,Y -556.384,Z 718.410,A 0.000,B 0.000,C 90.000,E1 289.758} C_DIS
LIN {X -0.112,Y -556.355,Z 718.410,A 0.000,B 0.000,C 90.000,E1 289.758} C_DIS
LIN {X 0.083,Y -555.552,Z 718.409,A 0.000,B 0.000,C 90.000,E1 289.577} C_DIS
LIN {X 0.221,Y -554.934,Z 718.407,A 0.000,B 0.000,C 90.000,E1 289.214} C_DIS
LIN {X 0.102,Y -554.763,Z 718.406,A 0.000,B 0.000,C 90.000,E1 289.087} C_DIS
LIN {X 0.011,Y -554.389,Z 718.400,A 0.000,B 0.000,C 90.000,E1 288.055} C_DIS
LIN {X 0.220,Y -553.612,Z 718.390,A 0.000,B 0.000,C 90.000,E1 286.079} C_DIS
LIN {X 0.258,Y -552.926,Z 718.379,A 0.000,B 0.000,C 90.000,E1 284.120} C_DIS
LIN {X 0.021,Y -552.316,Z 718.368,A 0.000,B 0.000,C 90.000,E1 282.187} C_DIS
LIN {X 0.198,Y -551.601,Z 718.358,A 0.000,B 0.000,C 90.000,E1 280.489} C_DIS
LIN {X 0.143,Y -550.971,Z 718.351,A 0.000,B 0.000,C 90.000,E1 279.095} C_DIS
LIN {X 0.211,Y -550.053,Z 718.340,A 0.000,B 0.000,C 90.000,E1 277.125} C_DIS
LIN {X 0.225,Y -549.275,Z 718.327,A 0.000,B 0.000,C 90.000,E1 274.878} C_DIS
LIN {X -0.142,Y -549.055,Z 718.323,A 0.000,B 0.000,C 90.000,E1 274.073} C_DIS
LIN {X 0.116,Y -548.715,Z 718.316,A 0.000,B 0.000,C 90.000,E1 272.922} C_DIS
LIN {X -0.123,Y -548.031,Z 718.307,A 0.000,B 0.000,C 90.000,E1 271.260} C_DIS
LIN {X 0.070,Y -547.456,Z 718.301,A 0.000,B 0.000,C 90.000,E1 270.115} C_DIS
LIN {X -0.205,Y -546.467,Z 718.291,A 0.000,B 0.000,C 90.000,E1 268.453} C_DIS
LIN {X 0.080,Y -545.404,Z 718.282,A 0.000,B 0.000,C 90.000,E1 266.731} C_DIS
LIN {X -0.265,Y -544.424,Z 718.274,A 0.000,B 0.000,C 90.000,E1 265.355} C_DIS
LIN {X 0.019,Y -543.162,Z 718.265,A 0.000,B 0.000,C 90.000,E1 263.628} C_DIS
LIN {X -0.272,Y -541.993,Z 718.257,A 0.000,B 0.000,C 90.000,E1 262.243} C_DIS
LIN {X 0.180,Y -540.278,Z 718.246,A 0.000,B 0.000,C 90.000,E1 260.208} C_DIS
LIN {X 0.125,Y -538.268,Z 718.233,A 0.000,B 0.000,C 90.000,E1 257.937} C_DIS
LIN {X 0.106,Y -536.749,Z 718.224,A 0.000,B 0.000,C 90.000,E1 256.228} C_DIS
LIN {X 0.001,Y -535.366,Z 718.216,A 0.000,B 0.000,C 90.000,E1 254.810} C_DIS
LIN {X 0.050,Y -533.616,Z 718.206,A 0.000,B 0.000,C 90.000,E1 253.087} C_DIS
LIN {X -0.298,Y -531.878,Z 718.197,A 0.000,B 0.000,C 90.000,E1 251.402} C_DIS
LIN {X -0.210,Y -530.496,Z 718.190,A 0.000,B 0.000,C 90.000,E1 250.242} C_DIS
LIN {X 0.229,Y -528.192,Z 718.181,A 0.000,B 0.000,C 90.000,E1 248.465} C_DIS
LIN {X -0.229,Y -526.546,Z 718.174,A 0.000,B 0.000,C 90.000,E1 247.358} C_DIS
LIN {X -0.026,Y -524.833,Z 718.168,A 0.000,B 0.000,C 90.000,E1 246.177} C_DIS
LIN {X 0.046,Y -522.448,Z 718.160,A 0.000,B 0.000,C 90.000,E1 244.717} C_DIS
LIN {X -0.064,Y -520.498,Z 718.153,A 0.000,B 0.000,C 90.000,E1 243.563} C_DIS
LIN {X 0.126,Y -518.925,Z 718.148,A 0.000,B 0.000,C 90.000,E1 242.666} C_DIS
LIN {X -0.014,Y -515.453,Z 718.138,A 0.000,B 0.000,C 90.000,E1 240.923} C_DIS
LIN {X 0.008,Y -513.116,Z 718.132,A 0.000,B 0.000,C 90.000,E1 239.744} C_DIS
LIN {X -0.204,Y -509.394,Z 718.122,A 0.000,B 0.000,C 90.000,E1 237.995} C_DIS
LIN {X 0.095,Y -505.071,Z 718.111,A 0.000,B 0.000,C 90.000,E1 235.881} C_DIS
LIN {X -0.037,Y -501.682,Z 718.102,A 0.000,B 0.000,C 90.000,E1 234.402} C_DIS
LIN {X 0.015,Y -499.536,Z 718.097,A 0.000,B 0.000,C 90.000,E1 233.497} C_DIS
LIN {X -0.233,Y -498.009,Z 718.094,A 0.000,B 0.000,C 90.000,E1 232.924} C_DIS
LIN {X -0.015,Y -491.863,Z 718.081,A 0.000,B 0.000,C 90.000,E1 230.481} C_DIS
LIN {X 0.187,Y -486.862,Z 718.069,A 0.000,B 0.000,C 90.000,E1 228.324} C_DIS
LIN {X -0.239,Y -484.067,Z 718.062,A 0.000,B 0.000,C 90.000,E1 227.148} C_DIS
LIN {X 0.111,Y -480.623,Z 718.053,A 0.000,B 0.000,C 90.000,E1 225.567} C_DIS
LIN {X 0.054,Y -475.249,Z 718.039,A 0.000,B 0.000,C 90.000,E1 223.095} C_DIS
LIN {X 0.003,Y -471.315,Z 718.029,A 0.000,B 0.000,C 90.000,E1 221.229} C_DIS
LIN {X 0.137,Y -467.925,Z 718.020,A 0.000,B 0.000,C 90.000,E1 219.644} C_DIS
LIN {X 0.147,Y -465.179,Z 718.013,A 0.000,B 0.000,C 90.000,E1 218.382} C_DIS
LIN {X 0.217,Y -458.868,Z 717.997,A 0.000,B 0.000,C 90.000,E1 215.518} C_DIS
LIN {X 0.103,Y -454.590,Z 717.985,A 0.000,B 0.000,C 90.000,E1 213.293} C_DIS
LIN {X 0.207,Y -451.556,Z 717.976,A 0.000,B 0.000,C 90.000,E1 211.671} C_DIS
LIN {X 0.024,Y -448.629,Z 717.967,A 0.000,B 0.000,C 90.000,E1 210.079} C_DIS
LIN {X 0.152,Y -443.877,Z 717.953,A 0.000,B 0.000,C 90.000,E1 207.462} C_DIS
LIN {X -0.046,Y -441.476,Z 717.945,A 0.000,B 0.000,C 90.000,E1 206.181} C_DIS
LIN {X -0.018,Y -437.894,Z 717.935,A 0.000,B 0.000,C 90.000,E1 204.207} C_DIS
LIN {X -0.096,Y -434.825,Z 717.925,A 0.000,B 0.000,C 90.000,E1 202.567} C_DIS
LIN {X 0.058,Y -431.114,Z 717.914,A 0.000,B 0.000,C 90.000,E1 200.556} C_DIS
LIN {X 0.133,Y -427.519,Z 717.903,A 0.000,B 0.000,C 90.000,E1 198.544} C_DIS
LIN {X 0.191,Y -424.414,Z 717.894,A 0.000,B 0.000,C 90.000,E1 196.858} C_DIS
LIN {X 0.064,Y -421.264,Z 717.884,A 0.000,B 0.000,C 90.000,E1 195.190} C_DIS
LIN {X -0.229,Y -418.259,Z 717.875,A 0.000,B 0.000,C 90.000,E1 193.536} C_DIS
LIN {X -0.128,Y -414.668,Z 717.864,A 0.000,B 0.000,C 90.000,E1 191.478} C_DIS
LIN {X 0.197,Y -411.063,Z 717.852,A 0.000,B 0.000,C 90.000,E1 189.378} C_DIS
LIN {X -0.122,Y -406.708,Z 717.837,A 0.000,B 0.000,C 90.000,E1 186.663} C_DIS
LIN {X -0.168,Y -403.603,Z 717.825,A 0.000,B 0.000,C 90.000,E1 184.588} C_DIS
LIN {X 0.046,Y -400.687,Z 717.814,A 0.000,B 0.000,C 90.000,E1 182.465} C_DIS
LIN {X 0.069,Y -397.374,Z 717.798,A 0.000,B 0.000,C 90.000,E1 179.656} C_DIS
LIN {X 0.004,Y -394.611,Z 717.783,A 0.000,B 0.000,C 90.000,E1 176.846} C_DIS
LIN {X -0.130,Y -392.417,Z 717.767,A 0.000,B 0.000,C 90.000,E1 174.033} C_DIS
LIN {X -0.170,Y -390.725,Z 717.751,A 0.000,B 0.000,C 90.000,E1 171.197} C_DIS
LIN {X -0.147,Y -389.718,Z 717.737,A 0.000,B 0.000,C 90.000,E1 168.701} C_DIS
LIN {X 0.143,Y -389.376,Z 717.731,A 0.000,B 0.000,C 90.000,E1 167.589} C_DIS
LIN {X 0.002,Y -388.582,Z 717.715,A 0.000,B 0.000,C 90.000,E1 164.755} C_DIS
LIN {X 0.160,Y -388.132,Z 717.699,A 0.000,B 0.000,C 90.000,E1 161.873} C_DIS
LIN {X 0.028,Y -387.949,Z 717.686,A 0.000,B 0.000,C 90.000,E1 159.390} C_DIS
LIN {X -0.030,Y -387.917,Z 717.670,A 0.000,B 0.000,C 90.000,E1 156.538} C_DIS
LIN {X -0.138,Y -388.031,Z 717.658,A 0.000,B 0.000,C 90.000,E1 154.409} C_DIS
LIN {X 0.085,Y -388.325,Z 717.646,A 0.000,B 0.000,C 90.000,E1 152.231} C_DIS
LIN {X -0.029,Y -388.672,Z 717.636,A 0.000,B 0.000,C 90.000,E1 150.461} C_DIS
LIN {X 0.036,Y -392.354,Z 717.600,A 0.000,B 0.000,C 90.000,E1 144.036} C_DIS
LIN {X 0.247,Y -395.402,Z 717.585,A 0.000,B 0.000,C 90.000,E1 141.170} C_DIS
LIN {X -0.032,Y -398.284,Z 717.573,A 0.000,B 0.000,C 90.000,E1 139.094} C_DIS
LIN {X 0.061,Y -400.957,Z 717.565,A 0.000,B 0.000,C 90.000,E1 137.676} C_DIS
LIN {X 0.107,Y -402.266,Z 717.562,A 0.000,B 0.000,C 90.000,E1 137.148} C_DIS
LIN {X 0.133,Y -404.302,Z 717.559,A 0.000,B 0.000,C 90.000,E1 136.620} C_DIS
LIN {X -0.122,Y -407.199,Z 717.556,A 0.000,B 0.000,C 90.000,E1 136.134} C_DIS
LIN {X -0.031,Y -411.541,Z 717.553,A 0.000,B 0.000,C 90.000,E1 135.567} C_DIS
LIN {X -0.222,Y -421.753,Z 717.547,A 0.000,B 0.000,C 90.000,E1 134.514} C_DIS
LIN {X 0.172,Y -433.818,Z 717.541,A 0.000,B 0.000,C 90.000,E1 133.299} C_DIS
LIN {X 0.092,Y -447.385,Z 717.534,A 0.000,B 0.000,C 90.000,E1 132.081} C_DIS
LIN {X -0.134,Y -462.080,Z 717.527,A 0.000,B 0.000,C 90.000,E1 130.782} C_DIS
LIN {X -0.118,Y -467.781,Z 717.524,A 0.000,B 0.000,C 90.000,E1 130.253} C_DIS
LIN {X 0.092,Y -476.419,Z 717.519,A 0.000,B 0.000,C 90.000,E1 129.402} C_DIS
LIN {X -0.100,Y -484.818,Z 717.514,A 0.000,B 0.000,C 90.000,E1 128.588} C_DIS
LIN {X -0.062,Y -494.225,Z 717.509,A 0.000,B 0.000,C 90.000,E1 127.604} C_DIS
LIN {X -0.043,Y -499.554,Z 717.506,A 0.000,B 0.000,C 90.000,E1 127.030} C_DIS
LIN {X -0.056,Y -505.796,Z 717.502,A 0.000,B 0.000,C 90.000,E1 126.297} C_DIS
LIN {X -0.068,Y -509.393,Z 717.499,A 0.000,B 0.000,C 90.000,E1 125.851} C_DIS
LIN {X 0.272,Y -513.758,Z 717.496,A 0.000,B 0.000,C 90.000,E1 125.231} C_DIS
LIN {X 0.009,Y -516.970,Z 717.493,A 0.000,B 0.000,C 90.000,E1 124.818} C_DIS
LIN {X 0.130,Y -521.722,Z 717.489,A 0.000,B 0.000,C 90.000,E1 124.072} C_DIS
LIN {X -0.106,Y -525.983,Z 717.485,A 0.000,B 0.000,C 90.000,E1 123.372} C_DIS
LIN {X 0.103,Y -529.923,Z 717.481,A 0.000,B 0.000,C 90.000,E1 122.625} C_DIS
LIN {X -0.230,Y -532.888,Z 717.478,A 0.000,B 0.000,C 90.000,E1 122.084} C_DIS
LIN {X 0.036,Y -537.500,Z 717.473,A 0.000,B 0.000,C 90.000,E1 121.052} C_DIS
LIN {X 0.076,Y -541.793,Z 717.467,A 0.000,B 0.000,C 90.000,E1 120.050} C_DIS
LIN {X -0.230,Y -546.418,Z 717.461,A 0.000,B 0.000,C 90.000,E1 118.949} C_DIS
LIN {X -0.230,Y -549.751,Z 717.456,A 0.000,B 0.000,C 90.000,E1 118.103} C_DIS
LIN {X -0.195,Y -552.827,Z 717.451,A 0.000,B 0.000,C 90.000,E1 117.257} C_DIS
LIN {X -0.131,Y -555.720,Z 717.447,A 0.000,B 0.000,C 90.000,E1 116.411} C_DIS
LIN {X 0.220,Y -558.323,Z 717.442,A 0.000,B 0.000,C 90.000,E1 115.540} C_DIS
LIN {X 0.103,Y -560.657,Z 717.437,A 0.000,B 0.000,C 90.000,E1 114.719} C_DIS
LIN {X 0.009,Y -562.666,Z 717.433,A 0.000,B 0.000,C 90.000,E1 113.898} C_DIS
LIN {X -0.067,Y -564.451,Z 717.428,A 0.000,B 0.000,C 90.000,E1 113.078} C_DIS
LIN {X -0.132,Y -565.960,Z 717.424,A 0.000,B 0.000,C 90.000,E1 112.259} C_DIS
LIN {X -0.116,Y -568.710,Z 717.414,A 0.000,B 0.000,C 90.000,E1 110.610} C_DIS
LIN {X -0.039,Y -571.331,Z 717.405,A 0.000,B 0.000,C 90.000,E1 108.960} C_DIS
LIN {X -0.083,Y -572.964,Z 717.399,A 0.000,B 0.000,C 90.000,E1 107.873} C_DIS
LIN {X -0.281,Y -575.302,Z 717.390,A 0.000,B 0.000,C 90.000,E1 106.260} C_DIS
LIN {X 0.125,Y -577.537,Z 717.381,A 0.000,B 0.000,C 90.000,E1 104.592} C_DIS
LIN {X 0.076,Y -579.312,Z 717.374,A 0.000,B 0.000,C 90.000,E1 103.244} C_DIS
LIN {X -0.037,Y -580.782,Z 717.368,A 0.000,B 0.000,C 90.000,E1 102.175} C_DIS
LIN {X -0.145,Y -582.626,Z 717.360,A 0.000,B 0.000,C 90.000,E1 100.838} C_DIS
LIN {X 0.225,Y -584.047,Z 717.354,A 0.000,B 0.000,C 90.000,E1 99.726} C_DIS
LIN {X 0.086,Y -585.634,Z 717.347,A 0.000,B 0.000,C 90.000,E1 98.398} C_DIS
LIN {X -0.111,Y -587.702,Z 717.336,A 0.000,B 0.000,C 90.000,E1 96.543} C_DIS
LIN {X 0.092,Y -588.775,Z 717.330,A 0.000,B 0.000,C 90.000,E1 95.454} C_DIS
LIN {X -0.017,Y -590.178,Z 717.323,A 0.000,B 0.000,C 90.000,E1 94.131} C_DIS
LIN {X 0.273,Y -591.200,Z 717.317,A 0.000,B 0.000,C 90.000,E1 93.037} C_DIS
LIN {X -0.226,Y -592.471,Z 717.308,A 0.000,B 0.000,C 90.000,E1 91.489} C_DIS
LIN {X 0.258,Y -593.327,Z 717.301,A 0.000,B 0.000,C 90.000,E1 90.115} C_DIS
LIN {X 0.165,Y -594.000,Z 717.293,A 0.000,B 0.000,C 90.000,E1 88.797} C_DIS
LIN {X 0.096,Y -594.482,Z 717.286,A 0.000,B 0.000,C 90.000,E1 87.478} C_DIS
LIN {X 0.035,Y -594.799,Z 717.279,A 0.000,B 0.000,C 90.000,E1 86.159} C_DIS
LIN {X 0.017,Y -594.954,Z 717.271,A 0.000,B 0.000,C 90.000,E1 84.837} C_DIS
LIN {X 0.112,Y -595.042,Z 717.267,A 0.000,B 0.000,C 90.000,E1 84.033} C_DIS
LIN {X -0.115,Y -595.052,Z 717.261,A 0.000,B 0.000,C 90.000,E1 82.996} C_DIS
LIN {X 0.014,Y -594.865,Z 717.254,A 0.000,B 0.000,C 90.000,E1 81.659} C_DIS
LIN {X 0.058,Y -594.456,Z 717.246,A 0.000,B 0.000,C 90.000,E1 80.330} C_DIS
LIN {X 0.183,Y -593.810,Z 717.239,A 0.000,B 0.000,C 90.000,E1 78.993} C_DIS
LIN {X -0.170,Y -592.982,Z 717.232,A 0.000,B 0.000,C 90.000,E1 77.701} C_DIS
LIN {X 0.043,Y -592.070,Z 717.224,A 0.000,B 0.000,C 90.000,E1 76.353} C_DIS
LIN {X 0.113,Y -591.207,Z 717.218,A 0.000,B 0.000,C 90.000,E1 75.283} C_DIS
LIN {X 0.177,Y -590.299,Z 717.212,A 0.000,B 0.000,C 90.000,E1 74.212} C_DIS
LIN {X -0.090,Y -589.065,Z 717.205,A 0.000,B 0.000,C 90.000,E1 72.906} C_DIS
LIN {X 0.111,Y -587.981,Z 717.199,A 0.000,B 0.000,C 90.000,E1 71.819} C_DIS
LIN {X -0.168,Y -586.149,Z 717.190,A 0.000,B 0.000,C 90.000,E1 70.242} C_DIS
LIN {X -0.014,Y -584.805,Z 717.184,A 0.000,B 0.000,C 90.000,E1 69.156} C_DIS
LIN {X 0.184,Y -582.925,Z 717.177,A 0.000,B 0.000,C 90.000,E1 67.794} C_DIS
LIN {X -0.047,Y -581.230,Z 717.171,A 0.000,B 0.000,C 90.000,E1 66.741} C_DIS
LIN {X -0.068,Y -579.309,Z 717.165,A 0.000,B 0.000,C 90.000,E1 65.665} C_DIS
LIN {X -0.109,Y -577.094,Z 717.159,A 0.000,B 0.000,C 90.000,E1 64.588} C_DIS
LIN {X -0.183,Y -574.632,Z 717.153,A 0.000,B 0.000,C 90.000,E1 63.512} C_DIS
LIN {X -0.035,Y -571.855,Z 717.147,A 0.000,B 0.000,C 90.000,E1 62.410} C_DIS
LIN {X -0.027,Y -569.580,Z 717.142,A 0.000,B 0.000,C 90.000,E1 61.591} C_DIS
LIN {X -0.275,Y -567.142,Z 717.138,A 0.000,B 0.000,C 90.000,E1 60.795} C_DIS
LIN {X 0.039,Y -563.429,Z 717.132,A 0.000,B 0.000,C 90.000,E1 59.665} C_DIS
LIN {X -0.066,Y -561.479,Z 717.128,A 0.000,B 0.000,C 90.000,E1 59.125} C_DIS
LIN {X 0.086,Y -558.241,Z 717.124,A 0.000,B 0.000,C 90.000,E1 58.280} C_DIS
LIN {X 0.130,Y -555.281,Z 717.120,A 0.000,B 0.000,C 90.000,E1 57.582} C_DIS
LIN {X -0.150,Y -552.053,Z 717.116,A 0.000,B 0.000,C 90.000,E1 56.914} C_DIS
LIN {X -0.158,Y -548.348,Z 717.112,A 0.000,B 0.000,C 90.000,E1 56.215} C_DIS
LIN {X 0.116,Y -543.383,Z 717.108,A 0.000,B 0.000,C 90.000,E1 55.341} C_DIS
LIN {X 0.318,Y -540.807,Z 717.105,A 0.000,B 0.000,C 90.000,E1 54.895} C_DIS
LIN {X 0.047,Y -537.085,Z 717.102,A 0.000,B 0.000,C 90.000,E1 54.356} C_DIS
LIN {X 0.061,Y -533.003,Z 717.099,A 0.000,B 0.000,C 90.000,E1 53.783} C_DIS
LIN {X 0.047,Y -528.391,Z 717.096,A 0.000,B 0.000,C 90.000,E1 53.210} C_DIS
LIN {X 0.021,Y -523.270,Z 717.092,A 0.000,B 0.000,C 90.000,E1 52.637} C_DIS
LIN {X 0.266,Y -519.244,Z 717.090,A 0.000,B 0.000,C 90.000,E1 52.190} C_DIS
LIN {X -0.078,Y -513.384,Z 717.087,A 0.000,B 0.000,C 90.000,E1 51.698} C_DIS
LIN {X 0.240,Y -507.190,Z 717.084,A 0.000,B 0.000,C 90.000,E1 51.170} C_DIS
LIN {X 0.114,Y -500.842,Z 717.082,A 0.000,B 0.000,C 90.000,E1 50.723} C_DIS
LIN {X 0.044,Y -492.819,Z 717.079,A 0.000,B 0.000,C 90.000,E1 50.194} C_DIS
LIN {X 0.101,Y -486.307,Z 717.077,A 0.000,B 0.000,C 90.000,E1 49.784} C_DIS
LIN {X 0.138,Y -468.205,Z 717.071,A 0.000,B 0.000,C 90.000,E1 48.690} C_DIS
LIN {X 0.013,Y -442.542,Z 717.062,A 0.000,B 0.000,C 90.000,E1 47.106} C_DIS
LIN {X -0.166,Y -423.161,Z 717.054,A 0.000,B 0.000,C 90.000,E1 45.810} C_DIS
LIN {X 0.008,Y -419.900,Z 717.053,A 0.000,B 0.000,C 90.000,E1 45.526} C_DIS
LIN {X -0.017,Y -419.876,Z 717.053,A 0.000,B 0.000,C 90.000,E1 45.526} C_DIS
LIN {X 0.149,Y -418.545,Z 717.049,A 0.000,B 0.000,C 90.000,E1 44.757} C_DIS
LIN {X -0.031,Y -408.987,Z 717.024,A 0.000,B 0.000,C 90.000,E1 40.334} C_DIS
LIN {X 0.117,Y -407.178,Z 717.018,A 0.000,B 0.000,C 90.000,E1 39.277} C_DIS
LIN {X -0.051,Y -407.056,Z 717.016,A 0.000,B 0.000,C 90.000,E1 38.955} C_DIS
LIN {X -0.093,Y -407.688,Z 716.995,A 0.000,B 0.000,C 90.000,E1 35.152} C_DIS
LIN {X -0.219,Y -408.199,Z 716.988,A 0.000,B 0.000,C 90.000,E1 33.785} C_DIS
LIN {X 0.070,Y -409.135,Z 716.976,A 0.000,B 0.000,C 90.000,E1 31.671} C_DIS
LIN {X -0.197,Y -410.559,Z 716.961,A 0.000,B 0.000,C 90.000,E1 28.949} C_DIS
LIN {X 0.172,Y -411.970,Z 716.947,A 0.000,B 0.000,C 90.000,E1 26.488} C_DIS
LIN {X -0.033,Y -413.979,Z 716.932,A 0.000,B 0.000,C 90.000,E1 23.770} C_DIS
LIN {X 0.118,Y -416.055,Z 716.919,A 0.000,B 0.000,C 90.000,E1 21.354} C_DIS
LIN {X 0.013,Y -418.111,Z 716.907,A 0.000,B 0.000,C 90.000,E1 19.322} C_DIS
LIN {X 0.239,Y -420.868,Z 716.894,A 0.000,B 0.000,C 90.000,E1 16.913} C_DIS
LIN {X -0.102,Y -423.888,Z 716.881,A 0.000,B 0.000,C 90.000,E1 14.592} C_DIS
LIN {X 0.081,Y -426.196,Z 716.872,A 0.000,B 0.000,C 90.000,E1 12.883} C_DIS
LIN {X 0.005,Y -429.415,Z 716.859,A 0.000,B 0.000,C 90.000,E1 10.546} C_DIS
LIN {X -0.179,Y -432.240,Z 716.848,A 0.000,B 0.000,C 90.000,E1 8.568} C_DIS
LIN {X -0.189,Y -434.141,Z 716.840,A 0.000,B 0.000,C 90.000,E1 7.239} C_DIS
LIN {X -0.085,Y -436.622,Z 716.831,A 0.000,B 0.000,C 90.000,E1 5.568} C_DIS
LIN {X 0.206,Y -441.878,Z 716.813,A 0.000,B 0.000,C 90.000,E1 2.236} C_DIS
LIN {X 0.169,Y -446.266,Z 716.799,A 0.000,B 0.000,C 90.000,E1 359.771} C_DIS
LIN {X 0.164,Y -449.986,Z 716.788,A 0.000,B 0.000,C 90.000,E1 357.822} C_DIS
LIN {X -0.016,Y -454.485,Z 716.776,A 0.000,B 0.000,C 90.000,E1 355.584} C_DIS
LIN {X -0.230,Y -458.545,Z 716.765,A 0.000,B 0.000,C 90.000,E1 353.685} C_DIS
LIN {X 0.188,Y -461.224,Z 716.758,A 0.000,B 0.000,C 90.000,E1 352.356} C_DIS
LIN {X 0.243,Y -465.059,Z 716.747,A 0.000,B 0.000,C 90.000,E1 350.443} C_DIS
LIN {X -0.079,Y -467.541,Z 716.740,A 0.000,B 0.000,C 90.000,E1 349.218} C_DIS
LIN {X 0.094,Y -469.914,Z 716.733,A 0.000,B 0.000,C 90.000,E1 347.937} C_DIS
LIN {X 0.049,Y -473.320,Z 716.723,A 0.000,B 0.000,C 90.000,E1 346.061} C_DIS
LIN {X 0.062,Y -475.675,Z 716.716,A 0.000,B 0.000,C 90.000,E1 344.810} C_DIS
LIN {X 0.189,Y -480.981,Z 716.700,A 0.000,B 0.000,C 90.000,E1 342.000} C_DIS
LIN {X -0.135,Y -485.610,Z 716.688,A 0.000,B 0.000,C 90.000,E1 339.880} C_DIS
LIN {X -0.125,Y -486.347,Z 716.686,A 0.000,B 0.000,C 90.000,E1 339.571} C_DIS
LIN {X -0.095,Y -488.210,Z 716.683,A 0.000,B 0.000,C 90.000,E1 338.954} C_DIS
LIN {X 0.167,Y -489.972,Z 716.681,A 0.000,B 0.000,C 90.000,E1 338.465} C_DIS
LIN {X 0.197,Y -491.516,Z 716.679,A 0.000,B 0.000,C 90.000,E1 338.156} C_DIS
LIN {X 0.231,Y -493.572,Z 716.677,A 0.000,B 0.000,C 90.000,E1 337.847} C_DIS
LIN {X -0.126,Y -496.633,Z 716.675,A 0.000,B 0.000,C 90.000,E1 337.539} C_DIS
LIN {X -0.044,Y -501.185,Z 716.673,A 0.000,B 0.000,C 90.000,E1 337.102} C_DIS
LIN {X 0.132,Y -508.276,Z 716.670,A 0.000,B 0.000,C 90.000,E1 336.538} C_DIS
LIN {X 0.004,Y -528.555,Z 716.662,A 0.000,B 0.000,C 90.000,E1 335.229} C_DIS
LIN {X 0.257,Y -537.856,Z 716.659,A 0.000,B 0.000,C 90.000,E1 334.588} C_DIS
LIN {X -0.167,Y -543.700,Z 716.657,A 0.000,B 0.000,C 90.000,E1 334.204} C_DIS
LIN {X 0.142,Y -549.448,Z 716.654,A 0.000,B 0.000,C 90.000,E1 333.717} C_DIS
LIN {X -0.001,Y -554.948,Z 716.651,A 0.000,B 0.000,C 90.000,E1 333.256} C_DIS
LIN {X 0.164,Y -560.424,Z 716.649,A 0.000,B 0.000,C 90.000,E1 332.743} C_DIS
LIN {X 0.169,Y -566.968,Z 716.645,A 0.000,B 0.000,C 90.000,E1 332.103} C_DIS
LIN {X 0.227,Y -573.297,Z 716.641,A 0.000,B 0.000,C 90.000,E1 331.435} C_DIS
LIN {X -0.028,Y -578.203,Z 716.638,A 0.000,B 0.000,C 90.000,E1 330.923} C_DIS
LIN {X -0.057,Y -588.830,Z 716.632,A 0.000,B 0.000,C 90.000,E1 329.715} C_DIS
LIN {X -0.343,Y -594.434,Z 716.628,A 0.000,B 0.000,C 90.000,E1 329.076} C_DIS
LIN {X -0.015,Y -601.882,Z 716.623,A 0.000,B 0.000,C 90.000,E1 328.122} C_DIS
LIN {X 0.189,Y -605.944,Z 716.620,A 0.000,B 0.000,C 90.000,E1 327.582} C_DIS
LIN {X -0.217,Y -612.743,Z 716.615,A 0.000,B 0.000,C 90.000,E1 326.707} C_DIS
LIN {X 0.019,Y -616.388,Z 716.612,A 0.000,B 0.000,C 90.000,E1 326.167} C_DIS
LIN {X 0.066,Y -622.463,Z 716.607,A 0.000,B 0.000,C 90.000,E1 325.261} C_DIS
LIN {X -0.334,Y -628.882,Z 716.601,A 0.000,B 0.000,C 90.000,E1 324.276} C_DIS
LIN {X 0.231,Y -634.897,Z 716.596,A 0.000,B 0.000,C 90.000,E1 323.210} C_DIS
LIN {X -0.126,Y -641.127,Z 716.589,A 0.000,B 0.000,C 90.000,E1 322.110} C_DIS
LIN {X 0.191,Y -645.104,Z 716.585,A 0.000,B 0.000,C 90.000,E1 321.331} C_DIS
LIN {X -0.024,Y -650.813,Z 716.579,A 0.000,B 0.000,C 90.000,E1 320.231} C_DIS
LIN {X 0.246,Y -655.558,Z 716.574,A 0.000,B 0.000,C 90.000,E1 319.218} C_DIS
LIN {X 0.153,Y -660.029,Z 716.568,A 0.000,B 0.000,C 90.000,E1 318.243} C_DIS
LIN {X -0.364,Y -663.219,Z 716.564,A 0.000,B 0.000,C 90.000,E1 317.553} C_DIS
LIN {X 0.084,Y -666.155,Z 716.560,A 0.000,B 0.000,C 90.000,E1 316.782} C_DIS
LIN {X 0.084,Y -669.847,Z 716.555,A 0.000,B 0.000,C 90.000,E1 315.810} C_DIS
LIN {X 0.137,Y -673.308,Z 716.549,A 0.000,B 0.000,C 90.000,E1 314.838} C_DIS
LIN {X 0.235,Y -676.548,Z 716.544,A 0.000,B 0.000,C 90.000,E1 313.866} C_DIS
LIN {X -0.057,Y -680.329,Z 716.537,A 0.000,B 0.000,C 90.000,E1 312.690} C_DIS
LIN {X -0.341,Y -683.224,Z 716.532,A 0.000,B 0.000,C 90.000,E1 311.757} C_DIS
LIN {X -0.024,Y -686.510,Z 716.525,A 0.000,B 0.000,C 90.000,E1 310.539} C_DIS
LIN {X 0.227,Y -688.323,Z 716.521,A 0.000,B 0.000,C 90.000,E1 309.806} C_DIS
LIN {X 0.023,Y -690.421,Z 716.516,A 0.000,B 0.000,C 90.000,E1 308.874} C_DIS
LIN {X -0.119,Y -691.829,Z 716.512,A 0.000,B 0.000,C 90.000,E1 308.177} C_DIS
LIN {X -0.173,Y -693.436,Z 716.507,A 0.000,B 0.000,C 90.000,E1 307.237} C_DIS
LIN {X 0.407,Y -695.188,Z 716.500,A 0.000,B 0.000,C 90.000,E1 306.011} C_DIS
LIN {X -0.019,Y -696.395,Z 716.495,A 0.000,B 0.000,C 90.000,E1 305.105} C_DIS
LIN {X 0.196,Y -697.632,Z 716.489,A 0.000,B 0.000,C 90.000,E1 303.913} C_DIS
LIN {X 0.380,Y -698.507,Z 716.483,A 0.000,B 0.000,C 90.000,E1 302.959} C_DIS
LIN {X -0.102,Y -699.668,Z 716.476,A 0.000,B 0.000,C 90.000,E1 301.592} C_DIS
LIN {X -0.258,Y -700.384,Z 716.470,A 0.000,B 0.000,C 90.000,E1 300.669} C_DIS
LIN {X -0.062,Y -700.716,Z 716.466,A 0.000,B 0.000,C 90.000,E1 299.951} C_DIS
LIN {X 0.010,Y -701.189,Z 716.457,A 0.000,B 0.000,C 90.000,E1 298.309} C_DIS
LIN {X -0.312,Y -701.961,Z 716.446,A 0.000,B 0.000,C 90.000,E1 296.232} C_DIS
LIN {X -0.135,Y -702.410,Z 716.440,A 0.000,B 0.000,C 90.000,E1 295.283} C_DIS
LIN {X 0.143,Y -702.382,Z 716.439,A 0.000,B 0.000,C 90.000,E1 295.027} C_DIS
LIN {X -0.231,Y -701.930,Z 716.437,A 0.000,B 0.000,C 90.000,E1 294.591} C_DIS
LIN {X 0.047,Y -701.261,Z 716.435,A 0.000,B 0.000,C 90.000,E1 294.335} C_DIS
LIN {X -0.329,Y -699.250,Z 716.433,A 0.000,B 0.000,C 90.000,E1 293.898} C_DIS
LIN {X -0.194,Y -698.524,Z 716.432,A 0.000,B 0.000,C 90.000,E1 293.770} C_DIS
LIN {X -0.060,Y -697.442,Z 716.431,A 0.000,B 0.000,C 90.000,E1 293.643} C_DIS
LIN {X 0.200,Y -694.315,Z 716.430,A 0.000,B 0.000,C 90.000,E1 293.387} C_DIS
LIN {X -0.062,Y -691.198,Z 716.429,A 0.000,B 0.000,C 90.000,E1 293.206} C_DIS
LIN {X 0.360,Y -689.476,Z 716.428,A 0.000,B 0.000,C 90.000,E1 293.078} C_DIS
LIN {X -0.124,Y -686.900,Z 716.428,A 0.000,B 0.000,C 90.000,E1 293.025} C_DIS
LIN {X 0.045,Y -684.722,Z 716.428,A 0.000,B 0.000,C 90.000,E1 292.950} C_DIS
LIN {X 0.087,Y -676.732,Z 716.427,A 0.000,B 0.000,C 90.000,E1 292.770} C_DIS
LIN {X -0.141,Y -659.243,Z 716.425,A 0.000,B 0.000,C 90.000,E1 292.567} C_DIS
LIN {X 0.095,Y -648.680,Z 716.424,A 0.000,B 0.000,C 90.000,E1 292.386} C_DIS
LIN {X 0.073,Y -638.823,Z 716.423,A 0.000,B 0.000,C 90.000,E1 292.206} C_DIS
LIN {X 0.207,Y -625.452,Z 716.422,A 0.000,B 0.000,C 90.000,E1 291.897} C_DIS
LIN {X -0.220,Y -611.967,Z 716.420,A 0.000,B 0.000,C 90.000,E1 291.589} C_DIS
LIN {X 0.233,Y -575.511,Z 716.414,A 0.000,B 0.000,C 90.000,E1 290.482} C_DIS
LIN {X 0.008,Y -570.140,Z 716.413,A 0.000,B 0.000,C 90.000,E1 290.355} C_DIS
LIN {X -0.253,Y -560.960,Z 716.411,A 0.000,B 0.000,C 90.000,E1 290.066} C_DIS
LIN {X 0.139,Y -559.255,Z 716.411,A 0.000,B 0.000,C 90.000,E1 289.939} C_DIS
LIN {X -0.015,Y -556.344,Z 716.410,A 0.000,B 0.000,C 90.000,E1 289.758} C_DIS
LIN {X -0.046,Y -556.319,Z 716.410,A 0.000,B 0.000,C 90.000,E1 289.758} C_DIS
LIN {X -0.251,Y -555.353,Z 716.409,A 0.000,B 0.000,C 90.000,E1 289.577} C_DIS
LIN {X 0.106,Y -554.764,Z 716.406,A 0.000,B 0.000,C 90.000,E1 289.087} C_DIS
LIN {X -0.167,Y -554.330,Z 716.400,A 0.000,B 0.000,C 90.000,E1 288.000} C_DIS
LIN {X 0.047,Y -553.557,Z 716.389,A 0.000,B 0.000,C 90.000,E1 286.024} C_DIS
LIN {X 0.088,Y -552.873,Z 716.378,A 0.000,B 0.000,C 90.000,E1 284.064} C_DIS
LIN {X -0.148,Y -552.344,Z 716.369,A 0.000,B 0.000,C 90.000,E1 282.411} C_DIS
LIN {X -0.099,Y -551.768,Z 716.361,A 0.000,B 0.000,C 90.000,E1 281.007} C_DIS
LIN {X -0.047,Y -551.014,Z 716.352,A 0.000,B 0.000,C 90.000,E1 279.321} C_DIS
LIN {X 0.013,Y -550.120,Z 716.341,A 0.000,B 0.000,C 90.000,E1 277.352} C_DIS
LIN {X 0.062,Y -549.259,Z 716.327,A 0.000,B 0.000,C 90.000,E1 274.821} C_DIS
LIN {X -0.172,Y -548.903,Z 716.319,A 0.000,B 0.000,C 90.000,E1 273.440} C_DIS
LIN {X 0.101,Y -548.359,Z 716.311,A 0.000,B 0.000,C 90.000,E1 272.007} C_DIS
LIN {X -0.186,Y -547.782,Z 716.303,A 0.000,B 0.000,C 90.000,E1 270.630} C_DIS
LIN {X 0.004,Y -547.128,Z 716.297,A 0.000,B 0.000,C 90.000,E1 269.484} C_DIS
LIN {X 0.240,Y -546.283,Z 716.289,A 0.000,B 0.000,C 90.000,E1 268.051} C_DIS
LIN {X -0.045,Y -545.243,Z 716.280,A 0.000,B 0.000,C 90.000,E1 266.388} C_DIS
LIN {X 0.189,Y -544.199,Z 716.272,A 0.000,B 0.000,C 90.000,E1 264.951} C_DIS
LIN {X -0.066,Y -542.941,Z 716.263,A 0.000,B 0.000,C 90.000,E1 263.280} C_DIS
LIN {X 0.177,Y -541.691,Z 716.255,A 0.000,B 0.000,C 90.000,E1 261.837} C_DIS
LIN {X 0.014,Y -540.235,Z 716.245,A 0.000,B 0.000,C 90.000,E1 260.151} C_DIS
LIN {X -0.113,Y -538.462,Z 716.234,A 0.000,B 0.000,C 90.000,E1 258.173} C_DIS
LIN {X 0.267,Y -537.424,Z 716.228,A 0.000,B 0.000,C 90.000,E1 256.992} C_DIS
LIN {X 0.044,Y -536.113,Z 716.220,A 0.000,B 0.000,C 90.000,E1 255.589} C_DIS
LIN {X 0.014,Y -535.020,Z 716.214,A 0.000,B 0.000,C 90.000,E1 254.448} C_DIS
LIN {X 0.250,Y -532.984,Z 716.203,A 0.000,B 0.000,C 90.000,E1 252.417} C_DIS
LIN {X -0.298,Y -531.527,Z 716.195,A 0.000,B 0.000,C 90.000,E1 251.040} C_DIS
LIN {X -0.027,Y -529.704,Z 716.187,A 0.000,B 0.000,C 90.000,E1 249.571} C_DIS
LIN {X 0.210,Y -527.719,Z 716.179,A 0.000,B 0.000,C 90.000,E1 248.103} C_DIS
LIN {X 0.118,Y -525.635,Z 716.170,A 0.000,B 0.000,C 90.000,E1 246.666} C_DIS
LIN {X -0.171,Y -523.826,Z 716.164,A 0.000,B 0.000,C 90.000,E1 245.537} C_DIS
LIN {X -0.109,Y -521.453,Z 716.156,A 0.000,B 0.000,C 90.000,E1 244.076} C_DIS
LIN {X 0.230,Y -519.368,Z 716.149,A 0.000,B 0.000,C 90.000,E1 242.871} C_DIS
LIN {X 0.067,Y -517.064,Z 716.143,A 0.000,B 0.000,C 90.000,E1 241.719} C_DIS
LIN {X 0.022,Y -514.201,Z 716.135,A 0.000,B 0.000,C 90.000,E1 240.255} C_DIS
LIN {X -0.066,Y -511.114,Z 716.127,A 0.000,B 0.000,C 90.000,E1 238.791} C_DIS
LIN {X 0.109,Y -507.363,Z 716.117,A 0.000,B 0.000,C 90.000,E1 236.993} C_DIS
LIN {X 0.119,Y -504.898,Z 716.110,A 0.000,B 0.000,C 90.000,E1 235.801} C_DIS
LIN {X -0.013,Y -501.527,Z 716.102,A 0.000,B 0.000,C 90.000,E1 234.322} C_DIS
LIN {X -0.083,Y -498.636,Z 716.095,A 0.000,B 0.000,C 90.000,E1 233.130} C_DIS
LIN {X -0.040,Y -494.664,Z 716.087,A 0.000,B 0.000,C 90.000,E1 231.618} C_DIS
LIN {X 0.071,Y -488.802,Z 716.073,A 0.000,B 0.000,C 90.000,E1 229.175} C_DIS
LIN {X 0.319,Y -484.607,Z 716.063,A 0.000,B 0.000,C 90.000,E1 227.310} C_DIS
LIN {X 0.124,Y -480.458,Z 716.053,A 0.000,B 0.000,C 90.000,E1 225.486} C_DIS
LIN {X 0.062,Y -475.066,Z 716.039,A 0.000,B 0.000,C 90.000,E1 223.014} C_DIS
LIN {X -0.083,Y -471.790,Z 716.030,A 0.000,B 0.000,C 90.000,E1 221.472} C_DIS
LIN {X 0.066,Y -468.424,Z 716.022,A 0.000,B 0.000,C 90.000,E1 219.886} C_DIS
LIN {X 0.139,Y -464.975,Z 716.013,A 0.000,B 0.000,C 90.000,E1 218.302} C_DIS
LIN {X -0.067,Y -458.700,Z 715.997,A 0.000,B 0.000,C 90.000,E1 215.471} C_DIS
LIN {X -0.277,Y -455.043,Z 715.986,A 0.000,B 0.000,C 90.000,E1 213.579} C_DIS
LIN {X 0.082,Y -452.028,Z 715.977,A 0.000,B 0.000,C 90.000,E1 211.926} C_DIS
LIN {X -0.097,Y -449.076,Z 715.969,A 0.000,B 0.000,C 90.000,E1 210.335} C_DIS
LIN {X 0.128,Y -445.447,Z 715.958,A 0.000,B 0.000,C 90.000,E1 208.359} C_DIS
LIN {X -0.049,Y -443.134,Z 715.950,A 0.000,B 0.000,C 90.000,E1 207.078} C_DIS
LIN {X -0.066,Y -440.709,Z 715.943,A 0.000,B 0.000,C 90.000,E1 205.771} C_DIS
LIN {X -0.087,Y -437.728,Z 715.934,A 0.000,B 0.000,C 90.000,E1 204.131} C_DIS
LIN {X -0.172,Y -435.290,Z 715.927,A 0.000,B 0.000,C 90.000,E1 202.823} C_DIS
LIN {X -0.032,Y -431.006,Z 715.914,A 0.000,B 0.000,C 90.000,E1 200.482} C_DIS
LIN {X 0.231,Y -427.982,Z 715.905,A 0.000,B 0.000,C 90.000,E1 198.779} C_DIS
LIN {X -0.043,Y -424.283,Z 715.893,A 0.000,B 0.000,C 90.000,E1 196.804} C_DIS
LIN {X 0.069,Y -419.963,Z 715.880,A 0.000,B 0.000,C 90.000,E1 194.426} C_DIS
LIN {X -0.101,Y -416.315,Z 715.869,A 0.000,B 0.000,C 90.000,E1 192.411} C_DIS
LIN {X 0.178,Y -413.930,Z 715.861,A 0.000,B 0.000,C 90.000,E1 191.007} C_DIS
LIN {X 0.006,Y -410.400,Z 715.850,A 0.000,B 0.000,C 90.000,E1 188.973} C_DIS
LIN {X 0.062,Y -406.647,Z 715.836,A 0.000,B 0.000,C 90.000,E1 186.549} C_DIS
LIN {X 0.018,Y -404.052,Z 715.827,A 0.000,B 0.000,C 90.000,E1 184.821} C_DIS
LIN {X -0.172,Y -400.675,Z 715.813,A 0.000,B 0.000,C 90.000,E1 182.407} C_DIS
LIN {X 0.193,Y -396.978,Z 715.796,A 0.000,B 0.000,C 90.000,E1 179.198} C_DIS
LIN {X 0.112,Y -394.306,Z 715.780,A 0.000,B 0.000,C 90.000,E1 176.388} C_DIS
LIN {X -0.003,Y -392.260,Z 715.764,A 0.000,B 0.000,C 90.000,E1 173.571} C_DIS
LIN {X 0.052,Y -391.070,Z 715.753,A 0.000,B 0.000,C 90.000,E1 171.432} C_DIS
LIN {X -0.011,Y -389.696,Z 715.733,A 0.000,B 0.000,C 90.000,E1 167.881} C_DIS
LIN {X -0.139,Y -388.814,Z 715.717,A 0.000,B 0.000,C 90.000,E1 165.046} C_DIS
LIN {X -0.143,Y -388.585,Z 715.711,A 0.000,B 0.000,C 90.000,E1 163.976} C_DIS
LIN {X -0.049,Y -388.317,Z 715.699,A 0.000,B 0.000,C 90.000,E1 161.819} C_DIS
LIN {X -0.182,Y -388.181,Z 715.685,A 0.000,B 0.000,C 90.000,E1 159.337} C_DIS
LIN {X -0.060,Y -388.188,Z 715.667,A 0.000,B 0.000,C 90.000,E1 156.102} C_DIS
LIN {X 0.015,Y -388.412,Z 715.653,A 0.000,B 0.000,C 90.000,E1 153.589} C_DIS
LIN {X 0.083,Y -388.756,Z 715.641,A 0.000,B 0.000,C 90.000,E1 151.435} C_DIS
LIN {X -0.100,Y -389.655,Z 715.624,A 0.000,B 0.000,C 90.000,E1 148.250} C_DIS
LIN {X -0.017,Y -393.261,Z 715.596,A 0.000,B 0.000,C 90.000,E1 143.256} C_DIS
LIN {X 0.026,Y -395.563,Z 715.584,A 0.000,B 0.000,C 90.000,E1 141.126} C_DIS
LIN {X 0.001,Y -398.384,Z 715.572,A 0.000,B 0.000,C 90.000,E1 139.013} C_DIS
LIN {X 0.015,Y -400.166,Z 715.566,A 0.000,B 0.000,C 90.000,E1 137.957} C_DIS
LIN {X 0.207,Y -401.676,Z 715.563,A 0.000,B 0.000,C 90.000,E1 137.229} C_DIS
LIN {X 0.026,Y -402.876,Z 715.561,A 0.000,B 0.000,C 90.000,E1 136.905} C_DIS
LIN {X 0.143,Y -404.111,Z 715.559,A 0.000,B 0.000,C 90.000,E1 136.539} C_DIS
LIN {X 0.057,Y -404.911,Z 715.558,A 0.000,B 0.000,C 90.000,E1 136.377} C_DIS
LIN {X -0.113,Y -406.859,Z 715.556,A 0.000,B 0.000,C 90.000,E1 136.053} C_DIS
LIN {X -0.197,Y -407.988,Z 715.555,A 0.000,B 0.000,C 90.000,E1 135.891} C_DIS
LIN {X 0.187,Y -410.697,Z 715.553,A 0.000,B 0.000,C 90.000,E1 135.486} C_DIS
LIN {X -0.167,Y -417.028,Z 715.549,A 0.000,B 0.000,C 90.000,E1 134.838} C_DIS
LIN {X 0.142,Y -430.437,Z 715.542,A 0.000,B 0.000,C 90.000,E1 133.461} C_DIS
LIN {X 0.028,Y -444.117,Z 715.535,A 0.000,B 0.000,C 90.000,E1 132.243} C_DIS
LIN {X -0.120,Y -460.622,Z 715.527,A 0.000,B 0.000,C 90.000,E1 130.782} C_DIS
LIN {X -0.113,Y -466.402,Z 715.524,A 0.000,B 0.000,C 90.000,E1 130.253} C_DIS
LIN {X -0.081,Y -474.994,Z 715.519,A 0.000,B 0.000,C 90.000,E1 129.439} C_DIS
LIN {X -0.091,Y -484.888,Z 715.514,A 0.000,B 0.000,C 90.000,E1 128.463} C_DIS
LIN {X 0.172,Y -494.459,Z 715.508,A 0.000,B 0.000,C 90.000,E1 127.443} C_DIS
LIN {X 0.225,Y -499.729,Z 715.505,A 0.000,B 0.000,C 90.000,E1 126.870} C_DIS
LIN {X 0.240,Y -504.647,Z 715.502,A 0.000,B 0.000,C 90.000,E1 126.297} C_DIS
LIN {X 0.040,Y -508.264,Z 715.499,A 0.000,B 0.000,C 90.000,E1 125.884} C_DIS
LIN {X -0.021,Y -512.771,Z 715.496,A 0.000,B 0.000,C 90.000,E1 125.311} C_DIS
LIN {X -0.183,Y -517.075,Z 715.493,A 0.000,B 0.000,C 90.000,E1 124.739} C_DIS
LIN {X 0.111,Y -521.006,Z 715.490,A 0.000,B 0.000,C 90.000,E1 124.119} C_DIS
LIN {X -0.129,Y -525.383,Z 715.486,A 0.000,B 0.000,C 90.000,E1 123.420} C_DIS
LIN {X 0.071,Y -529.411,Z 715.482,A 0.000,B 0.000,C 90.000,E1 122.673} C_DIS
LIN {X 0.182,Y -532.457,Z 715.478,A 0.000,B 0.000,C 90.000,E1 122.084} C_DIS
LIN {X -0.292,Y -537.174,Z 715.473,A 0.000,B 0.000,C 90.000,E1 121.131} C_DIS
LIN {X -0.117,Y -540.909,Z 715.468,A 0.000,B 0.000,C 90.000,E1 120.256} C_DIS
LIN {X 0.180,Y -546.218,Z 715.461,A 0.000,B 0.000,C 90.000,E1 118.949} C_DIS
LIN {X -0.059,Y -548.513,Z 715.458,A 0.000,B 0.000,C 90.000,E1 118.409} C_DIS
LIN {X 0.216,Y -552.681,Z 715.452,A 0.000,B 0.000,C 90.000,E1 117.257} C_DIS
LIN {X 0.033,Y -555.611,Z 715.447,A 0.000,B 0.000,C 90.000,E1 116.437} C_DIS
LIN {X 0.128,Y -558.252,Z 715.442,A 0.000,B 0.000,C 90.000,E1 115.591} C_DIS
LIN {X 0.006,Y -560.654,Z 715.438,A 0.000,B 0.000,C 90.000,E1 114.771} C_DIS
LIN {X -0.091,Y -562.708,Z 715.433,A 0.000,B 0.000,C 90.000,E1 113.951} C_DIS
LIN {X -0.170,Y -564.529,Z 715.428,A 0.000,B 0.000,C 90.000,E1 113.131} C_DIS
LIN {X 0.072,Y -566.081,Z 715.424,A 0.000,B 0.000,C 90.000,E1 112.280} C_DIS
LIN {X -0.226,Y -568.875,Z 715.415,A 0.000,B 0.000,C 90.000,E1 110.663} C_DIS
LIN {X 0.014,Y -571.962,Z 715.404,A 0.000,B 0.000,C 90.000,E1 108.725} C_DIS
LIN {X -0.018,Y -573.580,Z 715.398,A 0.000,B 0.000,C 90.000,E1 107.638} C_DIS
LIN {X -0.198,Y -575.955,Z 715.389,A 0.000,B 0.000,C 90.000,E1 106.024} C_DIS
LIN {X 0.223,Y -578.190,Z 715.380,A 0.000,B 0.000,C 90.000,E1 104.356} C_DIS
LIN {X 0.071,Y -580.757,Z 715.369,A 0.000,B 0.000,C 90.000,E1 102.479} C_DIS
LIN {X -0.252,Y -582.971,Z 715.360,A 0.000,B 0.000,C 90.000,E1 100.894} C_DIS
LIN {X 0.263,Y -584.758,Z 715.353,A 0.000,B 0.000,C 90.000,E1 99.500} C_DIS
LIN {X 0.230,Y -586.328,Z 715.346,A 0.000,B 0.000,C 90.000,E1 98.163} C_DIS
LIN {X -0.271,Y -588.138,Z 715.337,A 0.000,B 0.000,C 90.000,E1 96.606} C_DIS
LIN {X -0.183,Y -588.986,Z 715.332,A 0.000,B 0.000,C 90.000,E1 95.796} C_DIS
LIN {X -0.099,Y -590.661,Z 715.323,A 0.000,B 0.000,C 90.000,E1 94.188} C_DIS
LIN {X 0.198,Y -591.696,Z 715.317,A 0.000,B 0.000,C 90.000,E1 93.094} C_DIS
LIN {X 0.301,Y -592.978,Z 715.308,A 0.000,B 0.000,C 90.000,E1 91.489} C_DIS
LIN {X 0.201,Y -593.858,Z 715.301,A 0.000,B 0.000,C 90.000,E1 90.172} C_DIS
LIN {X -0.104,Y -594.412,Z 715.295,A 0.000,B 0.000,C 90.000,E1 89.141} C_DIS
LIN {X -0.165,Y -594.947,Z 715.288,A 0.000,B 0.000,C 90.000,E1 87.822} C_DIS
LIN {X -0.213,Y -595.300,Z 715.281,A 0.000,B 0.000,C 90.000,E1 86.502} C_DIS
LIN {X -0.218,Y -595.494,Z 715.273,A 0.000,B 0.000,C 90.000,E1 85.179} C_DIS
LIN {X -0.217,Y -595.573,Z 715.266,A 0.000,B 0.000,C 90.000,E1 83.856} C_DIS
LIN {X 0.159,Y -595.550,Z 715.260,A 0.000,B 0.000,C 90.000,E1 82.761} C_DIS
LIN {X 0.218,Y -595.339,Z 715.253,A 0.000,B 0.000,C 90.000,E1 81.432} C_DIS
LIN {X 0.078,Y -594.977,Z 715.247,A 0.000,B 0.000,C 90.000,E1 80.387} C_DIS
LIN {X 0.214,Y -594.316,Z 715.239,A 0.000,B 0.000,C 90.000,E1 79.050} C_DIS
LIN {X 0.151,Y -593.297,Z 715.230,A 0.000,B 0.000,C 90.000,E1 77.465} C_DIS
LIN {X -0.206,Y -592.332,Z 715.223,A 0.000,B 0.000,C 90.000,E1 76.172} C_DIS
LIN {X 0.027,Y -591.669,Z 715.219,A 0.000,B 0.000,C 90.000,E1 75.353} C_DIS
LIN {X -0.059,Y -590.474,Z 715.211,A 0.000,B 0.000,C 90.000,E1 74.031} C_DIS
LIN {X -0.323,Y -589.196,Z 715.204,A 0.000,B 0.000,C 90.000,E1 72.725} C_DIS
LIN {X -0.118,Y -588.044,Z 715.198,A 0.000,B 0.000,C 90.000,E1 71.638} C_DIS
LIN {X -0.065,Y -586.502,Z 715.191,A 0.000,B 0.000,C 90.000,E1 70.296} C_DIS
LIN {X 0.098,Y -585.110,Z 715.185,A 0.000,B 0.000,C 90.000,E1 69.209} C_DIS
LIN {X -0.101,Y -583.602,Z 715.179,A 0.000,B 0.000,C 90.000,E1 68.156} C_DIS
LIN {X 0.219,Y -581.947,Z 715.173,A 0.000,B 0.000,C 90.000,E1 67.050} C_DIS
LIN {X -0.028,Y -580.037,Z 715.167,A 0.000,B 0.000,C 90.000,E1 65.997} C_DIS
LIN {X -0.067,Y -577.881,Z 715.161,A 0.000,B 0.000,C 90.000,E1 64.921} C_DIS
LIN {X 0.119,Y -575.429,Z 715.155,A 0.000,B 0.000,C 90.000,E1 63.819} C_DIS
LIN {X 0.176,Y -573.410,Z 715.150,A 0.000,B 0.000,C 90.000,E1 62.999} C_DIS
LIN {X -0.303,Y -571.235,Z 715.146,A 0.000,B 0.000,C 90.000,E1 62.231} C_DIS
LIN {X -0.208,Y -567.986,Z 715.140,A 0.000,B 0.000,C 90.000,E1 61.129} C_DIS
LIN {X 0.206,Y -566.252,Z 715.136,A 0.000,B 0.000,C 90.000,E1 60.539} C_DIS
LIN {X -0.073,Y -563.451,Z 715.132,A 0.000,B 0.000,C 90.000,E1 59.744} C_DIS
LIN {X -0.180,Y -561.481,Z 715.129,A 0.000,B 0.000,C 90.000,E1 59.203} C_DIS
LIN {X 0.263,Y -558.196,Z 715.124,A 0.000,B 0.000,C 90.000,E1 58.329} C_DIS
LIN {X 0.012,Y -555.223,Z 715.120,A 0.000,B 0.000,C 90.000,E1 57.661} C_DIS
LIN {X 0.031,Y -551.913,Z 715.117,A 0.000,B 0.000,C 90.000,E1 56.962} C_DIS
LIN {X -0.281,Y -548.148,Z 715.113,A 0.000,B 0.000,C 90.000,E1 56.294} C_DIS
LIN {X 0.128,Y -543.957,Z 715.109,A 0.000,B 0.000,C 90.000,E1 55.548} C_DIS
LIN {X 0.189,Y -540.480,Z 715.106,A 0.000,B 0.000,C 90.000,E1 54.975} C_DIS
LIN {X 0.228,Y -536.694,Z 715.102,A 0.000,B 0.000,C 90.000,E1 54.402} C_DIS
LIN {X -0.073,Y -532.511,Z 715.099,A 0.000,B 0.000,C 90.000,E1 53.863} C_DIS
LIN {X -0.091,Y -527.786,Z 715.096,A 0.000,B 0.000,C 90.000,E1 53.290} C_DIS
LIN {X 0.044,Y -523.943,Z 715.094,A 0.000,B 0.000,C 90.000,E1 52.844} C_DIS
LIN {X 0.200,Y -518.511,Z 715.091,A 0.000,B 0.000,C 90.000,E1 52.271} C_DIS
LIN {X -0.026,Y -514.144,Z 715.088,A 0.000,B 0.000,C 90.000,E1 51.904} C_DIS
LIN {X -0.042,Y -507.982,Z 715.086,A 0.000,B 0.000,C 90.000,E1 51.412} C_DIS
LIN {X -0.197,Y -501.551,Z 715.083,A 0.000,B 0.000,C 90.000,E1 50.964} C_DIS
LIN {X -0.075,Y -495.082,Z 715.081,A 0.000,B 0.000,C 90.000,E1 50.517} C_DIS
LIN {X 0.018,Y -490.202,Z 715.079,A 0.000,B 0.000,C 90.000,E1 50.194} C_DIS
LIN {X 0.091,Y -472.053,Z 715.073,A 0.000,B 0.000,C 90.000,E1 49.094} C_DIS
LIN {X 0.142,Y -465.316,Z 715.071,A 0.000,B 0.000,C 90.000,E1 48.690} C_DIS
LIN {X 0.011,Y -446.230,Z 715.064,A 0.000,B 0.000,C 90.000,E1 47.514} C_DIS
LIN {X 0.091,Y -423.484,Z 715.056,A 0.000,B 0.000,C 90.000,E1 45.972} C_DIS
LIN {X -0.001,Y -420.275,Z 715.054,A 0.000,B 0.000,C 90.000,E1 45.729} C_DIS
LIN {X -0.030,Y -420.241,Z 715.054,A 0.000,B 0.000,C 90.000,E1 45.729} C_DIS
LIN {X 0.178,Y -418.715,Z 715.049,A 0.000,B 0.000,C 90.000,E1 44.838} C_DIS
LIN {X -0.152,Y -409.784,Z 715.026,A 0.000,B 0.000,C 90.000,E1 40.782} C_DIS
LIN {X -0.073,Y -407.617,Z 715.020,A 0.000,B 0.000,C 90.000,E1 39.564} C_DIS
LIN {X 0.160,Y -407.452,Z 715.019,A 0.000,B 0.000,C 90.000,E1 39.358} C_DIS
LIN {X 0.130,Y -408.143,Z 714.995,A 0.000,B 0.000,C 90.000,E1 35.025} C_DIS
LIN {X 0.015,Y -408.670,Z 714.987,A 0.000,B 0.000,C 90.000,E1 33.658} C_DIS
LIN {X 0.051,Y -409.466,Z 714.977,A 0.000,B 0.000,C 90.000,E1 31.926} C_DIS
LIN {X 0.072,Y -411.084,Z 714.960,A 0.000,B 0.000,C 90.000,E1 28.821} C_DIS
LIN {X 0.164,Y -412.297,Z 714.949,A 0.000,B 0.000,C 90.000,E1 26.744} C_DIS
LIN {X -0.029,Y -414.233,Z 714.934,A 0.000,B 0.000,C 90.000,E1 24.027} C_DIS
LIN {X 0.048,Y -416.593,Z 714.918,A 0.000,B 0.000,C 90.000,E1 21.280} C_DIS
LIN {X 0.042,Y -418.291,Z 714.909,A 0.000,B 0.000,C 90.000,E1 19.577} C_DIS
LIN {X 0.112,Y -420.584,Z 714.898,A 0.000,B 0.000,C 90.000,E1 17.528} C_DIS
LIN {X 0.055,Y -422.632,Z 714.888,A 0.000,B 0.000,C 90.000,E1 15.843} C_DIS
LIN {X -0.012,Y -425.279,Z 714.877,A 0.000,B 0.000,C 90.000,E1 13.828} C_DIS
LIN {X 0.018,Y -427.106,Z 714.869,A 0.000,B 0.000,C 90.000,E1 12.479} C_DIS
LIN {X -0.135,Y -429.859,Z 714.858,A 0.000,B 0.000,C 90.000,E1 10.489} C_DIS
LIN {X 0.004,Y -432.198,Z 714.849,A 0.000,B 0.000,C 90.000,E1 8.803} C_DIS
LIN {X 0.054,Y -434.102,Z 714.842,A 0.000,B 0.000,C 90.000,E1 7.466} C_DIS
LIN {X 0.152,Y -436.531,Z 714.832,A 0.000,B 0.000,C 90.000,E1 5.796} C_DIS
LIN {X -0.124,Y -441.124,Z 714.816,A 0.000,B 0.000,C 90.000,E1 2.865} C_DIS
LIN {X 0.057,Y -443.941,Z 714.807,A 0.000,B 0.000,C 90.000,E1 1.203} C_DIS
LIN {X 0.008,Y -447.718,Z 714.795,A 0.000,B 0.000,C 90.000,E1 359.141} C_DIS
LIN {X 0.171,Y -450.210,Z 714.788,A 0.000,B 0.000,C 90.000,E1 357.822} C_DIS
LIN {X -0.169,Y -454.054,Z 714.777,A 0.000,B 0.000,C 90.000,E1 355.927} C_DIS
LIN {X 0.069,Y -458.044,Z 714.767,A 0.000,B 0.000,C 90.000,E1 353.970} C_DIS
LIN {X -0.031,Y -460.767,Z 714.760,A 0.000,B 0.000,C 90.000,E1 352.704} C_DIS
LIN {X 0.173,Y -462.667,Z 714.754,A 0.000,B 0.000,C 90.000,E1 351.724} C_DIS
LIN {X -0.128,Y -466.452,Z 714.744,A 0.000,B 0.000,C 90.000,E1 349.859} C_DIS
LIN {X 0.032,Y -468.915,Z 714.737,A 0.000,B 0.000,C 90.000,E1 348.578} C_DIS
LIN {X -0.239,Y -471.177,Z 714.730,A 0.000,B 0.000,C 90.000,E1 347.353} C_DIS
LIN {X 0.143,Y -475.200,Z 714.717,A 0.000,B 0.000,C 90.000,E1 345.117} C_DIS
LIN {X 0.185,Y -477.463,Z 714.711,A 0.000,B 0.000,C 90.000,E1 343.866} C_DIS
LIN {X 0.068,Y -481.716,Z 714.698,A 0.000,B 0.000,C 90.000,E1 341.710} C_DIS
LIN {X -0.081,Y -486.360,Z 714.687,A 0.000,B 0.000,C 90.000,E1 339.571} C_DIS
LIN {X -0.050,Y -488.028,Z 714.683,A 0.000,B 0.000,C 90.000,E1 338.954} C_DIS
LIN {X -0.004,Y -490.089,Z 714.680,A 0.000,B 0.000,C 90.000,E1 338.337} C_DIS
LIN {X 0.028,Y -491.807,Z 714.678,A 0.000,B 0.000,C 90.000,E1 337.975} C_DIS
LIN {X -0.085,Y -493.930,Z 714.676,A 0.000,B 0.000,C 90.000,E1 337.667} C_DIS
LIN {X -0.044,Y -496.444,Z 714.674,A 0.000,B 0.000,C 90.000,E1 337.358} C_DIS
